C05456=1026.653,394.249,352.776,173.191,48.323,159.736
C05457=1026.645,394.003,352.820,173.181,48.321,159.734
C05458=1026.634,393.757,352.863,173.171,48.319,159.732
C05459=1026.625,393.511,352.907,173.161,48.317,159.730
C05460=1026.615,393.265,352.950,173.152,48.315,159.728
C05461=1026.606,393.019,352.994,173.141,48.312,159.726
C05462=1026.597,392.773,353.037,173.132,48.310,159.724
C05463=1026.586,392.527,353.080,173.121,48.309,159.722
C05464=1026.578,392.281,353.123,173.112,48.307,159.720
C05465=1026.568,392.035,353.167,173.102,48.304,159.718
C05466=1026.558,391.789,353.209,173.092,48.303,159.716
C05467=1026.549,391.543,353.253,173.082,48.301,159.714
C05468=1026.539,391.297,353.296,173.073,48.299,159.712
C05469=1026.530,391.051,353.338,173.063,48.297,159.711
C05470=1026.521,390.805,353.382,173.053,48.295,159.709
C05471=1026.511,390.559,353.425,173.044,48.293,159.707
C05472=1026.502,390.312,353.468,173.034,48.291,159.705
C05473=1026.493,390.067,353.511,173.024,48.289,159.703
C05474=1026.483,389.821,353.554,173.014,48.287,159.701
C05475=1026.474,389.575,353.597,173.005,48.285,159.699
C05476=1026.465,389.329,353.640,172.996,48.283,159.697
C05477=1026.455,389.083,353.683,172.987,48.282,159.696
C05478=1026.446,388.837,353.725,172.976,48.280,159.694
C05479=1026.437,388.590,353.768,172.967,48.278,159.692
C05480=1026.428,388.344,353.811,172.957,48.276,159.690
C05481=1026.418,388.097,353.853,172.948,48.275,159.688
C05482=1026.409,387.852,353.895,172.939,48.273,159.686
C05483=1026.400,387.606,353.938,172.930,48.271,159.685
C05484=1026.391,387.360,353.981,172.920,48.269,159.683
C05485=1026.381,387.113,354.024,172.910,48.268,159.681
C05486=1026.372,386.867,354.065,172.901,48.266,159.679
C05487=1026.363,386.621,354.108,172.892,48.264,159.677
C05488=1026.354,386.376,354.150,172.883,48.263,159.676
C05489=1026.344,386.128,354.192,172.873,48.261,159.674
C05490=1026.335,385.883,354.235,172.864,48.259,159.672
C05491=1026.326,385.636,354.276,172.855,48.258,159.671
C05492=1026.317,385.391,354.319,172.846,48.256,159.669
C05493=1026.307,385.144,354.361,172.837,48.255,159.667
C05494=1026.299,384.897,354.403,172.828,48.253,159.665
C05495=1026.289,384.651,354.445,172.818,48.252,159.664
C05496=1026.280,384.405,354.487,172.809,48.250,159.662
C05497=1026.271,384.159,354.528,172.800,48.248,159.660
C05498=1026.262,383.913,354.571,172.791,48.247,159.659
C05499=1026.253,383.667,354.613,172.782,48.245,159.657
C05500=1026.244,383.420,354.654,172.773,48.244,159.655
C05501=1026.235,383.174,354.696,172.764,48.242,159.654
C05502=1026.226,382.927,354.738,172.755,48.241,159.652
C05503=1026.218,382.681,354.779,172.746,48.240,159.650
C05504=1026.209,382.435,354.821,172.737,48.238,159.649
C05505=1026.199,382.189,354.862,172.728,48.237,159.647
C05506=1026.190,381.942,354.904,172.719,48.235,159.645
C05507=1026.181,381.696,354.946,172.710,48.234,159.644
C05508=1026.172,381.456,354.987,172.702,48.233,159.642
C05509=1026.163,381.216,355.028,172.693,48.231,159.641
C05510=1026.155,380.976,355.068,172.684,48.230,159.639
C05511=1026.146,380.736,355.109,172.676,48.229,159.638
C05512=1026.138,380.496,355.149,172.667,48.227,159.636
C05513=1026.129,380.257,355.189,172.659,48.226,159.634
C05514=1026.120,380.017,355.230,172.650,48.225,159.633
C05515=1026.112,379.776,355.270,172.641,48.223,159.631
C05516=1026.104,379.530,355.311,172.632,48.222,159.630
C05517=1026.095,379.284,355.353,172.624,48.220,159.628
C05518=1026.086,379.037,355.394,172.616,48.220,159.627
C05519=1026.077,378.790,355.435,172.607,48.218,159.625
C05520=1026.068,378.545,355.476,172.598,48.217,159.623
C05521=1026.059,378.298,355.517,172.590,48.216,159.622
C05522=1026.051,378.052,355.559,172.581,48.214,159.620
C05523=1026.042,377.805,355.600,172.572,48.213,159.619
C05524=1026.034,377.559,355.641,172.564,48.212,159.617
C05525=1026.025,377.312,355.682,172.555,48.211,159.616
C05526=1026.017,377.066,355.724,172.547,48.210,159.614
C05527=1026.008,376.819,355.765,172.539,48.208,159.613
C05528=1025.999,376.573,355.805,172.530,48.207,159.611
C05529=1025.990,376.327,355.846,172.521,48.206,159.610
C05530=1025.982,376.080,355.887,172.512,48.205,159.608
C05531=1025.972,375.833,355.928,172.505,48.204,159.607
C05532=1025.964,375.587,355.968,172.496,48.203,159.605
C05533=1025.955,375.340,356.009,172.488,48.201,159.604
C05534=1025.947,375.094,356.049,172.479,48.201,159.602
C05535=1025.937,374.847,356.090,172.470,48.200,159.601
C05536=1025.929,374.601,356.131,172.463,48.199,159.600
C05537=1025.921,374.354,356.172,172.454,48.198,159.598
C05538=1025.912,374.108,356.212,172.445,48.197,159.597
C05539=1025.903,373.861,356.253,172.438,48.196,159.595
C05540=1025.895,373.615,356.293,172.429,48.195,159.594
C05541=1025.886,373.368,356.334,172.421,48.193,159.592
C05542=1025.877,373.122,356.374,172.413,48.193,159.591
C05543=1025.869,372.875,356.415,172.405,48.191,159.589
C05544=1025.861,372.628,356.455,172.396,48.191,159.588
C05545=1025.852,372.382,356.495,172.388,48.190,159.587
C05546=1025.844,372.135,356.536,172.380,48.189,159.585
C05547=1025.835,371.889,356.576,172.371,48.188,159.584
C05548=1025.827,371.642,356.616,172.364,48.187,159.583
C05549=1025.818,371.396,356.656,172.355,48.187,159.581
C05550=1025.810,371.149,356.697,172.348,48.185,159.580
C05551=1025.802,370.903,356.737,172.340,48.184,159.578
C05552=1025.793,370.656,356.777,172.331,48.184,159.577
C05553=1025.785,370.409,356.817,172.324,48.183,159.576
C05554=1025.776,370.163,356.857,172.315,48.182,159.574
C05555=1025.768,369.916,356.897,172.308,48.181,159.573
C05556=1025.760,369.670,356.937,172.299,48.180,159.572
C05557=1025.751,369.423,356.977,172.292,48.180,159.571
C05558=1025.743,369.176,357.018,172.283,48.179,159.569
C05559=1025.735,368.930,357.057,172.276,48.178,159.568
C05560=1025.727,368.683,357.097,172.268,48.177,159.566
C05561=1025.718,368.437,357.137,172.259,48.177,159.565
C05562=1025.710,368.190,357.176,172.252,48.176,159.564
C05563=1025.701,367.943,357.216,172.243,48.175,159.563
C05564=1025.693,367.696,357.256,172.236,48.175,159.561
C05565=1025.685,367.449,357.295,172.228,48.173,159.560
C05566=1025.676,367.203,357.335,172.220,48.173,159.559
C05567=1025.668,366.956,357.374,172.213,48.173,159.558
C05568=1025.660,366.727,357.411,172.205,48.172,159.556
C05569=1025.652,366.498,357.448,172.198,48.171,159.555
C05570=1025.645,366.269,357.485,172.190,48.171,159.554
C05571=1025.637,366.039,357.521,172.183,48.170,159.553
C05572=1025.629,365.809,357.558,172.176,48.170,159.552
C05573=1025.622,365.580,357.595,172.169,48.170,159.551
C05574=1025.614,365.351,357.631,172.162,48.169,159.549
C05575=1025.607,365.122,357.668,172.155,48.168,159.548
C05576=1025.598,364.875,357.707,172.147,48.168,159.547
C05577=1025.590,364.629,357.747,172.139,48.167,159.546
C05578=1025.582,364.381,357.785,172.132,48.166,159.545
C05579=1025.573,364.135,357.825,172.124,48.166,159.543
C05580=1025.566,363.888,357.864,172.116,48.166,159.542
C05581=1025.557,363.641,357.904,172.109,48.165,159.541
C05582=1025.549,363.394,357.942,172.101,48.164,159.540
C05583=1025.540,363.147,357.982,172.094,48.164,159.539
C05584=1025.533,362.901,358.022,172.086,48.163,159.537
C05585=1025.525,362.654,358.060,172.079,48.163,159.536
C05586=1025.517,362.407,358.099,172.071,48.163,159.535
C05587=1025.509,362.160,358.138,172.064,48.162,159.534
C05588=1025.500,361.914,358.177,172.056,48.161,159.533
C05589=1025.493,361.666,358.216,172.048,48.161,159.531
C05590=1025.485,361.420,358.255,172.041,48.161,159.530
C05591=1025.477,361.173,358.294,172.034,48.160,159.529
C05592=1025.468,360.926,358.333,172.026,48.160,159.528
C05593=1025.460,360.679,358.372,172.019,48.159,159.527
C05594=1025.453,360.433,358.411,172.012,48.159,159.526
C05595=1025.445,360.186,358.450,172.004,48.159,159.525
C05596=1025.437,359.939,358.489,171.997,48.159,159.524
C05597=1025.428,359.691,358.527,171.989,48.158,159.522
C05598=1025.421,359.445,358.566,171.982,48.158,159.521
C05599=1025.412,359.198,358.605,171.975,48.158,159.520
C05600=1025.404,358.951,358.643,171.968,48.158,159.519
C05601=1025.397,358.705,358.682,171.959,48.157,159.518
C05602=1025.388,358.458,358.720,171.952,48.157,159.517
C05603=1025.380,358.210,358.758,171.945,48.157,159.516
C05604=1025.372,357.964,358.796,171.938,48.157,159.515
C05605=1025.364,357.717,358.835,171.931,48.157,159.514
C05606=1025.356,357.470,358.873,171.924,48.156,159.513
C05607=1025.348,357.223,358.912,171.916,48.156,159.512
C05608=1025.340,356.976,358.951,171.909,48.156,159.511
C05609=1025.333,356.729,358.989,171.902,48.155,159.509
C05610=1025.324,356.482,359.027,171.895,48.155,159.508
C05611=1025.317,356.235,359.066,171.888,48.155,159.507
C05612=1025.308,355.989,359.104,171.880,48.155,159.506
C05613=1025.301,355.741,359.141,171.873,48.155,159.505
C05614=1025.293,355.494,359.180,171.866,48.155,159.504
C05615=1025.285,355.248,359.218,171.859,48.155,159.503
C05616=1025.277,355.000,359.257,171.852,48.155,159.502
C05617=1025.270,354.753,359.294,171.844,48.155,159.501
C05618=1025.262,354.506,359.333,171.837,48.155,159.500
C05619=1025.253,354.260,359.370,171.830,48.155,159.499
C05620=1025.246,354.013,359.408,171.823,48.155,159.498
C05621=1025.238,353.766,359.447,171.816,48.155,159.497
C05622=1025.230,353.519,359.484,171.809,48.155,159.496
C05623=1025.222,353.272,359.522,171.802,48.155,159.495
C05624=1025.214,353.024,359.560,171.795,48.154,159.494
C05625=1025.206,352.778,359.597,171.788,48.154,159.493
C05626=1025.198,352.530,359.635,171.781,48.154,159.492
C05627=1025.191,352.284,359.673,171.774,48.154,159.491
C05628=1025.183,352.058,359.708,171.768,48.155,159.490
C05629=1025.176,351.832,359.742,171.761,48.155,159.489
C05630=1025.170,351.606,359.777,171.755,48.154,159.488
C05631=1025.162,351.380,359.811,171.749,48.155,159.488
C05632=1025.155,351.154,359.846,171.743,48.155,159.487
C05633=1025.147,350.928,359.880,171.737,48.155,159.486
C05634=1025.141,350.702,359.914,171.730,48.155,159.485
C05635=1025.134,350.476,359.949,171.724,48.155,159.484
C05636=1025.126,350.229,359.986,171.717,48.155,159.483
C05637=1025.119,349.982,360.024,171.710,48.155,159.482
C05638=1025.111,349.734,360.061,171.704,48.156,159.481
C05639=1025.103,349.488,360.099,171.696,48.156,159.480
C05640=1025.096,349.241,360.137,171.689,48.155,159.479
C05641=1025.088,348.993,360.174,171.683,48.156,159.479
C05642=1025.080,348.747,360.211,171.676,48.156,159.478
C05643=1025.073,348.499,360.249,171.670,48.156,159.477
C05644=1025.065,348.252,360.286,171.663,48.156,159.476
C05645=1025.057,348.005,360.323,171.656,48.156,159.475
C05646=1025.050,347.758,360.361,171.649,48.157,159.474
C05647=1025.042,347.511,360.398,171.642,48.157,159.473
C05648=1025.035,347.264,360.435,171.636,48.157,159.472
C05649=1025.027,347.017,360.472,171.629,48.158,159.471
C05650=1025.019,346.769,360.509,171.622,48.158,159.470
C05651=1025.012,346.522,360.546,171.616,48.158,159.470
C05652=1025.004,346.275,360.583,171.609,48.158,159.469
C05653=1024.997,346.028,360.621,171.602,48.159,159.468
C05654=1024.988,345.781,360.658,171.596,48.159,159.467
C05655=1024.981,345.533,360.695,171.589,48.159,159.466
C05656=1024.973,345.286,360.732,171.582,48.160,159.465
C05657=1024.965,345.039,360.768,171.576,48.160,159.465
C05658=1024.958,344.792,360.805,171.570,48.161,159.464
C05659=1024.950,344.545,360.842,171.562,48.161,159.463
C05660=1024.943,344.297,360.879,171.556,48.161,159.462
C05661=1024.936,344.051,360.916,171.549,48.162,159.461
C05662=1024.928,343.804,360.953,171.543,48.162,159.460
C05663=1024.921,343.556,360.989,171.537,48.163,159.460
C05664=1024.913,343.310,361.026,171.530,48.162,159.459
C05665=1024.905,343.062,361.063,171.523,48.163,159.458
C05666=1024.898,342.815,361.100,171.517,48.163,159.457
C05667=1024.890,342.567,361.136,171.511,48.164,159.456
C05668=1024.883,342.320,361.172,171.504,48.164,159.455
C05669=1024.876,342.073,361.210,171.497,48.165,159.455
C05670=1024.868,341.825,361.246,171.491,48.165,159.454
C05671=1024.860,341.579,361.283,171.485,48.166,159.453
C05672=1024.854,341.332,361.320,171.478,48.166,159.452
C05673=1024.846,341.084,361.356,171.471,48.167,159.451
C05674=1024.838,340.837,361.392,171.466,48.167,159.451
C05675=1024.831,340.590,361.430,171.459,48.168,159.450
C05676=1024.824,340.343,361.465,171.452,48.168,159.449
C05677=1024.816,340.095,361.502,171.446,48.169,159.448
C05678=1024.809,339.848,361.538,171.440,48.169,159.448
C05679=1024.802,339.600,361.575,171.433,48.170,159.447
C05680=1024.794,339.353,361.612,171.427,48.171,159.446
C05681=1024.787,339.107,361.647,171.421,48.171,159.445
C05682=1024.779,338.859,361.684,171.414,48.172,159.445
C05683=1024.771,338.612,361.720,171.408,48.172,159.444
C05684=1024.764,338.365,361.756,171.401,48.173,159.443
C05685=1024.756,338.118,361.792,171.396,48.174,159.442
C05686=1024.749,337.870,361.828,171.389,48.174,159.442
C05687=1024.741,337.622,361.864,171.383,48.176,159.441
C05688=1024.735,337.395,361.898,171.377,48.176,159.440
C05689=1024.728,337.168,361.930,171.372,48.177,159.440
C05690=1024.721,336.940,361.964,171.366,48.177,159.439
C05691=1024.714,336.713,361.997,171.359,48.178,159.438
C05692=1024.708,336.485,362.030,171.354,48.178,159.438
C05693=1024.700,336.257,362.063,171.348,48.179,159.437
C05694=1024.694,336.030,362.096,171.343,48.179,159.436
C05695=1024.687,335.803,362.129,171.337,48.180,159.436
C05696=1024.680,335.555,362.164,171.331,48.181,159.435
C05697=1024.673,335.307,362.201,171.324,48.182,159.434
C05698=1024.666,335.061,362.237,171.319,48.182,159.434
C05699=1024.658,334.813,362.273,171.312,48.184,159.433
C05700=1024.651,334.565,362.309,171.306,48.184,159.432
C05701=1024.644,334.318,362.344,171.300,48.185,159.432
C05702=1024.636,334.071,362.381,171.293,48.186,159.431
C05703=1024.629,333.824,362.416,171.288,48.186,159.430
C05704=1024.622,333.576,362.452,171.281,48.187,159.429
C05705=1024.615,333.329,362.487,171.275,48.188,159.429
C05706=1024.607,333.081,362.523,171.270,48.189,159.428
C05707=1024.600,332.834,362.558,171.263,48.190,159.427
C05708=1024.592,332.587,362.594,171.258,48.190,159.427
C05709=1024.585,332.340,362.629,171.251,48.192,159.426
C05710=1024.578,332.093,362.665,171.245,48.193,159.426
C05711=1024.571,331.845,362.701,171.239,48.193,159.425
C05712=1024.563,331.598,362.735,171.233,48.194,159.424
C05713=1024.556,331.350,362.771,171.227,48.195,159.424
C05714=1024.549,331.103,362.806,171.221,48.196,159.423
C05715=1024.542,330.855,362.842,171.215,48.198,159.423
C05716=1024.535,330.607,362.877,171.209,48.198,159.422
C05717=1024.527,330.361,362.912,171.203,48.199,159.421
C05718=1024.520,330.113,362.948,171.197,48.200,159.421
C05719=1024.513,329.866,362.983,171.191,48.201,159.420
C05720=1024.506,329.618,363.018,171.185,48.202,159.419
C05721=1024.498,329.371,363.054,171.179,48.203,159.419
C05722=1024.491,329.124,363.089,171.174,48.204,159.418
C05723=1024.484,328.876,363.124,171.167,48.205,159.418
C05724=1024.477,328.628,363.160,171.161,48.206,159.417
C05725=1024.470,328.381,363.195,171.156,48.207,159.416
C05726=1024.463,328.134,363.229,171.149,48.208,159.416
C05727=1024.456,327.886,363.264,171.144,48.209,159.415
C05728=1024.448,327.638,363.300,171.138,48.210,159.415
C05729=1024.441,327.392,363.336,171.132,48.211,159.414
C05730=1024.435,327.144,363.371,171.126,48.212,159.414
C05731=1024.427,326.897,363.405,171.120,48.213,159.413
C05732=1024.419,326.649,363.440,171.114,48.215,159.412
C05733=1024.412,326.401,363.475,171.109,48.215,159.412
C05734=1024.405,326.154,363.509,171.103,48.217,159.411
C05735=1024.397,325.907,363.544,171.097,48.218,159.411
C05736=1024.390,325.659,363.579,171.091,48.219,159.410
C05737=1024.383,325.412,363.613,171.085,48.220,159.410
C05738=1024.375,325.165,363.648,171.079,48.222,159.409
C05739=1024.369,324.917,363.682,171.073,48.223,159.409
C05740=1024.361,324.670,363.717,171.068,48.224,159.408
C05741=1024.353,324.422,363.752,171.062,48.226,159.408
C05742=1024.347,324.174,363.786,171.056,48.227,159.407
C05743=1024.339,323.927,363.820,171.050,48.228,159.406
C05744=1024.332,323.680,363.855,171.045,48.229,159.406
C05745=1024.325,323.432,363.889,171.039,48.231,159.405
C05746=1024.318,323.185,363.924,171.034,48.232,159.405
C05747=1024.311,322.937,363.958,171.027,48.233,159.404
C05748=1024.304,322.707,363.990,171.022,48.235,159.404
C05749=1024.297,322.477,364.023,171.017,48.236,159.404
C05750=1024.290,322.248,364.054,171.011,48.237,159.403
C05751=1024.284,322.018,364.086,171.006,48.238,159.403
C05752=1024.277,321.788,364.119,171.001,48.240,159.402
C05753=1024.270,321.558,364.150,170.996,48.240,159.402
C05754=1024.264,321.328,364.182,170.991,48.242,159.401
C05755=1024.258,321.099,364.214,170.986,48.243,159.401
C05756=1024.251,320.851,364.248,170.980,48.245,159.400
C05757=1024.243,320.604,364.282,170.974,48.245,159.400
C05758=1024.236,320.356,364.316,170.968,48.247,159.399
C05759=1024.230,320.108,364.351,170.963,48.248,159.399
C05760=1024.222,319.861,364.385,170.957,48.250,159.398
C05761=1024.215,319.614,364.419,170.952,48.251,159.398
C05762=1024.208,319.366,364.453,170.946,48.252,159.397
C05763=1024.201,319.118,364.488,170.940,48.254,159.397
C05764=1024.194,318.871,364.522,170.935,48.256,159.397
C05765=1024.187,318.623,364.556,170.929,48.257,159.396
C05766=1024.180,318.375,364.590,170.924,48.258,159.396
C05767=1024.173,318.129,364.624,170.918,48.260,159.395
C05768=1024.167,317.881,364.659,170.912,48.261,159.395
C05769=1024.160,317.633,364.693,170.907,48.263,159.394
C05770=1024.152,317.385,364.726,170.901,48.264,159.394
C05771=1024.146,317.137,364.761,170.896,48.265,159.393
C05772=1024.138,316.890,364.795,170.890,48.267,159.393
C05773=1024.132,316.643,364.829,170.885,48.269,159.393
C05774=1024.125,316.396,364.863,170.880,48.270,159.392
C05775=1024.118,316.148,364.897,170.874,48.271,159.392
C05776=1024.111,315.900,364.931,170.868,48.273,159.391
C05777=1024.104,315.652,364.965,170.863,48.274,159.391
C05778=1024.098,315.405,364.999,170.857,48.276,159.390
C05779=1024.091,315.157,365.033,170.852,48.278,159.390
C05780=1024.083,314.910,365.066,170.846,48.279,159.390
C05781=1024.077,314.662,365.101,170.841,48.281,159.389
C05782=1024.070,314.415,365.134,170.836,48.282,159.389
C05783=1024.063,314.167,365.168,170.830,48.284,159.388
C05784=1024.056,313.919,365.202,170.825,48.285,159.388
C05785=1024.050,313.672,365.236,170.820,48.287,159.387
C05786=1024.043,313.425,365.270,170.814,48.288,159.387
C05787=1024.036,313.177,365.304,170.809,48.290,159.387
C05788=1024.030,312.930,365.338,170.804,48.291,159.386
C05789=1024.023,312.681,365.371,170.798,48.293,159.386
C05790=1024.016,312.434,365.404,170.793,48.295,159.385
C05791=1024.009,312.187,365.438,170.788,48.296,159.385
C05792=1024.003,311.939,365.472,170.783,48.298,159.385
C05793=1023.996,311.692,365.506,170.777,48.299,159.384
C05794=1023.989,311.444,365.540,170.771,48.301,159.384
C05795=1023.983,311.196,365.572,170.766,48.302,159.384
C05796=1023.976,310.948,365.607,170.760,48.304,159.383
C05797=1023.970,310.701,365.640,170.755,48.306,159.383
C05798=1023.962,310.454,365.674,170.750,48.307,159.382
C05799=1023.955,310.205,365.707,170.744,48.309,159.382
C05800=1023.949,309.958,365.740,170.740,48.311,159.382
C05801=1023.941,309.711,365.773,170.735,48.313,159.381
C05802=1023.935,309.463,365.806,170.728,48.315,159.381
C05803=1023.928,309.215,365.840,170.724,48.317,159.381
C05804=1023.920,308.967,365.872,170.718,48.319,159.380
C05805=1023.914,308.720,365.905,170.713,48.321,159.380
C05806=1023.907,308.472,365.939,170.708,48.322,159.380
C05807=1023.900,308.225,365.971,170.702,48.324,159.379
C05808=1023.893,307.997,366.001,170.697,48.326,159.379
C05809=1023.886,307.770,366.032,170.693,48.327,159.379
C05810=1023.880,307.543,366.062,170.689,48.330,159.379
C05811=1023.874,307.316,366.092,170.684,48.331,159.378
C05812=1023.868,307.089,366.122,170.678,48.333,159.378
C05813=1023.861,306.861,366.152,170.674,48.335,159.378
C05814=1023.855,306.634,366.183,170.669,48.336,159.377
C05815=1023.849,306.407,366.213,170.664,48.338,159.377
C05816=1023.842,306.159,366.246,170.659,48.340,159.377
C05817=1023.835,305.911,366.278,170.654,48.342,159.377
C05818=1023.827,305.664,366.312,170.648,48.344,159.376
C05819=1023.821,305.416,366.345,170.644,48.346,159.376
C05820=1023.814,305.169,366.377,170.639,48.347,159.376
C05821=1023.807,304.921,366.410,170.633,48.350,159.375
C05822=1023.801,304.673,366.443,170.628,48.352,159.375
C05823=1023.793,304.425,366.475,170.623,48.354,159.375
C05824=1023.787,304.177,366.508,170.617,48.356,159.375
C05825=1023.781,303.930,366.541,170.612,48.357,159.374
C05826=1023.773,303.682,366.573,170.608,48.360,159.374
C05827=1023.767,303.434,366.606,170.602,48.362,159.374
C05828=1023.760,303.186,366.639,170.597,48.364,159.373
C05829=1023.753,302.939,366.671,170.592,48.366,159.373
C05830=1023.747,302.691,366.704,170.587,48.368,159.373
C05831=1023.740,302.444,366.736,170.581,48.370,159.373
C05832=1023.733,302.195,366.769,170.577,48.372,159.372
C05833=1023.726,301.948,366.802,170.572,48.374,159.372
C05834=1023.719,301.701,366.834,170.567,48.376,159.372
C05835=1023.712,301.452,366.867,170.561,48.378,159.372
C05836=1023.706,301.205,366.900,170.557,48.380,159.371
C05837=1023.699,300.957,366.932,170.552,48.382,159.371
C05838=1023.692,300.709,366.965,170.547,48.384,159.371
C05839=1023.685,300.461,366.997,170.541,48.386,159.371
C05840=1023.679,300.214,367.029,170.536,48.388,159.370
C05841=1023.673,299.966,367.062,170.532,48.391,159.370
C05842=1023.666,299.719,367.094,170.527,48.393,159.370
C05843=1023.659,299.470,367.127,170.521,48.394,159.370
C05844=1023.653,299.222,367.159,170.516,48.397,159.369
C05845=1023.646,298.975,367.191,170.512,48.399,159.369
C05846=1023.640,298.727,367.224,170.507,48.401,159.369
C05847=1023.633,298.480,367.256,170.501,48.403,159.369
C05848=1023.626,298.231,367.289,170.496,48.406,159.369
C05849=1023.620,297.984,367.321,170.492,48.408,159.368
C05850=1023.613,297.736,367.354,170.487,48.409,159.368
C05851=1023.607,297.488,367.386,170.482,48.411,159.368
C05852=1023.600,297.241,367.418,170.476,48.414,159.368
C05853=1023.593,296.993,367.451,170.472,48.416,159.367
C05854=1023.587,296.745,367.483,170.467,48.418,159.367
C05855=1023.580,296.498,367.515,170.462,48.420,159.367
C05856=1023.574,296.249,367.547,170.458,48.422,159.367
C05857=1023.567,296.001,367.580,170.452,48.425,159.367
C05858=1023.561,295.753,367.611,170.447,48.427,159.366
C05859=1023.554,295.506,367.644,170.442,48.429,159.366
C05860=1023.547,295.258,367.676,170.438,48.431,159.366
C05861=1023.541,295.010,367.708,170.433,48.433,159.366
C05862=1023.535,294.763,367.741,170.427,48.436,159.366
C05863=1023.528,294.515,367.772,170.423,48.438,159.365
C05864=1023.522,294.267,367.804,170.418,48.440,159.365
C05865=1023.515,294.019,367.837,170.413,48.442,159.365
C05866=1023.509,293.771,367.869,170.408,48.445,159.365
C05867=1023.502,293.524,367.901,170.404,48.447,159.365
C05868=1023.497,293.305,367.929,170.399,48.450,159.365
C05869=1023.491,293.086,367.957,170.395,48.452,159.365
C05870=1023.485,292.868,367.985,170.391,48.454,159.364
C05871=1023.480,292.650,368.013,170.386,48.456,159.364
C05872=1023.473,292.430,368.041,170.383,48.458,159.364
C05873=1023.467,292.212,368.069,170.378,48.460,159.364
C05874=1023.462,291.994,368.097,170.373,48.462,159.364
C05875=1023.456,291.775,368.124,170.370,48.464,159.364
C05876=1023.450,291.527,368.156,170.365,48.467,159.364
C05877=1023.443,291.280,368.188,170.359,48.469,159.363
C05878=1023.437,291.032,368.220,170.355,48.471,159.363
C05879=1023.430,290.784,368.251,170.350,48.474,159.363
C05880=1023.423,290.536,368.283,170.346,48.476,159.363
C05881=1023.416,290.288,368.314,170.341,48.478,159.363
C05882=1023.410,290.040,368.346,170.336,48.481,159.363
C05883=1023.403,289.792,368.377,170.331,48.483,159.363
C05884=1023.396,289.545,368.409,170.327,48.486,159.363
C05885=1023.390,289.297,368.440,170.322,48.488,159.362
C05886=1023.384,289.048,368.472,170.317,48.491,159.362
C05887=1023.377,288.801,368.503,170.312,48.494,159.362
C05888=1023.370,288.553,368.535,170.307,48.497,159.362
C05889=1023.363,288.305,368.566,170.303,48.499,159.362
C05890=1023.357,288.057,368.598,170.298,48.501,159.362
C05891=1023.351,287.810,368.629,170.294,48.504,159.362
C05892=1023.344,287.561,368.659,170.288,48.507,159.362
C05893=1023.337,287.313,368.691,170.284,48.509,159.361
C05894=1023.331,287.065,368.722,170.279,48.512,159.361
C05895=1023.324,286.817,368.754,170.275,48.514,159.361
C05896=1023.317,286.569,368.785,170.270,48.517,159.361
C05897=1023.311,286.321,368.816,170.265,48.519,159.361
C05898=1023.305,286.073,368.848,170.260,48.522,159.361
C05899=1023.299,285.826,368.879,170.256,48.525,159.361
C05900=1023.292,285.578,368.910,170.251,48.527,159.361
C05901=1023.285,285.330,368.942,170.247,48.530,159.361
C05902=1023.278,285.082,368.972,170.242,48.533,159.361
C05903=1023.271,284.834,369.003,170.237,48.535,159.361
C05904=1023.266,284.586,369.034,170.232,48.538,159.361
C05905=1023.259,284.338,369.065,170.228,48.541,159.361
C05906=1023.252,284.090,369.097,170.223,48.543,159.361
C05907=1023.246,283.841,369.127,170.219,48.546,159.360
C05908=1023.238,283.594,369.158,170.214,48.548,159.360
C05909=1023.232,283.346,369.189,170.209,48.552,159.360
C05910=1023.226,283.098,369.220,170.205,48.554,159.360
C05911=1023.219,282.850,369.251,170.200,48.557,159.360
C05912=1023.213,282.602,369.282,170.196,48.559,159.360
C05913=1023.207,282.354,369.312,170.191,48.562,159.360
C05914=1023.199,282.106,369.343,170.186,48.565,159.360
C05915=1023.193,281.858,369.374,170.182,48.568,159.360
C05916=1023.186,281.610,369.405,170.177,48.571,159.360
C05917=1023.180,281.362,369.436,170.173,48.574,159.360
C05918=1023.174,281.114,369.467,170.168,48.576,159.360
C05919=1023.166,280.866,369.497,170.164,48.579,159.360
C05920=1023.161,280.618,369.528,170.158,48.582,159.360
C05921=1023.154,280.370,369.559,170.154,48.585,159.360
C05922=1023.147,280.122,369.590,170.150,48.587,159.360
C05923=1023.142,279.874,369.620,170.145,48.590,159.360
C05924=1023.135,279.626,369.652,170.141,48.593,159.360
C05925=1023.128,279.378,369.682,170.137,48.596,159.360
C05926=1023.122,279.130,369.712,170.132,48.599,159.360
C05927=1023.115,278.882,369.744,170.127,48.602,159.360
C05928=1023.110,278.669,369.770,170.123,48.604,159.360
C05929=1023.104,278.457,369.796,170.120,48.606,159.360
C05930=1023.099,278.245,369.822,170.115,48.609,159.360
C05931=1023.093,278.032,369.848,170.112,48.611,159.360
C05932=1023.088,277.820,369.875,170.108,48.614,159.360
C05933=1023.083,277.608,369.901,170.104,48.616,159.359
C05934=1023.077,277.396,369.927,170.101,48.619,159.360
C05935=1023.071,277.182,369.953,170.096,48.621,159.360
C05936=1023.065,276.934,369.984,170.092,48.624,159.360
C05937=1023.058,276.686,370.014,170.088,48.627,159.360
C05938=1023.052,276.438,370.044,170.083,48.630,159.360
C05939=1023.045,276.190,370.074,170.079,48.633,159.360
C05940=1023.039,275.943,370.105,170.074,48.637,159.360
C05941=1023.032,275.695,370.135,170.069,48.639,159.360
C05942=1023.026,275.447,370.166,170.065,48.642,159.360
C05943=1023.020,275.198,370.197,170.061,48.645,159.360
C05944=1023.013,274.950,370.227,170.056,48.648,159.360
C05945=1023.007,274.702,370.257,170.052,48.651,159.360
C05946=1023.000,274.454,370.287,170.047,48.654,159.360
C05947=1022.994,274.206,370.317,170.043,48.657,159.360
C05948=1022.987,273.958,370.347,170.038,48.660,159.360
C05949=1022.981,273.710,370.377,170.034,48.664,159.360
C05950=1022.974,273.462,370.407,170.030,48.666,159.360
C05951=1022.968,273.214,370.438,170.026,48.669,159.360
C05952=1022.962,272.965,370.468,170.021,48.672,159.360
C05953=1022.955,272.718,370.498,170.016,48.676,159.360
C05954=1022.948,272.469,370.528,170.012,48.679,159.360
C05955=1022.942,272.222,370.559,170.007,48.681,159.360
C05956=1022.936,271.974,370.588,170.003,48.685,159.360
C05957=1022.930,271.725,370.618,169.999,48.688,159.360
C05958=1022.923,271.477,370.648,169.995,48.691,159.360
C05959=1022.917,271.229,370.679,169.991,48.694,159.360
C05960=1022.910,270.981,370.709,169.985,48.697,159.360
C05961=1022.904,270.732,370.739,169.981,48.701,159.360
C05962=1022.897,270.485,370.768,169.977,48.703,159.360
C05963=1022.892,270.237,370.799,169.973,48.707,159.361
C05964=1022.885,269.988,370.828,169.969,48.710,159.361
C05965=1022.878,269.741,370.858,169.965,48.713,159.361
C05966=1022.872,269.492,370.889,169.960,48.716,159.361
C05967=1022.866,269.244,370.918,169.955,48.720,159.361
C05968=1022.859,268.996,370.947,169.951,48.723,159.361
C05969=1022.853,268.748,370.978,169.947,48.726,159.361
C05970=1022.846,268.500,371.007,169.942,48.729,159.361
C05971=1022.839,268.252,371.037,169.938,48.732,159.361
C05972=1022.834,268.003,371.067,169.934,48.735,159.361
C05973=1022.827,267.756,371.097,169.930,48.739,159.361
C05974=1022.820,267.507,371.126,169.925,48.743,159.361
C05975=1022.814,267.259,371.156,169.921,48.745,159.361
C05976=1022.808,267.011,371.185,169.917,48.749,159.362
C05977=1022.801,266.763,371.216,169.912,48.752,159.362
C05978=1022.795,266.515,371.245,169.908,48.755,159.362
C05979=1022.789,266.267,371.275,169.904,48.759,159.362
C05980=1022.782,266.018,371.304,169.900,48.762,159.362
C05981=1022.776,265.770,371.334,169.895,48.765,159.362
C05982=1022.769,265.522,371.363,169.891,48.769,159.362
C05983=1022.763,265.274,371.392,169.887,48.772,159.362
C05984=1022.757,265.026,371.423,169.882,48.775,159.362
C05985=1022.750,264.777,371.452,169.878,48.779,159.362
C05986=1022.744,264.529,371.481,169.874,48.782,159.363
C05987=1022.737,264.281,371.511,169.869,48.786,159.363
C05988=1022.726,263.861,371.560,169.863,48.791,159.363
C05989=1022.721,263.651,371.585,169.859,48.794,159.363
C05990=1022.716,263.441,371.610,169.855,48.797,159.363
C05991=1022.710,263.231,371.635,169.852,48.800,159.363
C05992=1022.705,263.020,371.660,169.848,48.803,159.363
C05993=1022.699,262.810,371.685,169.845,48.806,159.363
C05994=1022.694,262.600,371.709,169.842,48.809,159.364
C05995=1022.687,262.352,371.739,169.836,48.812,159.364
C05996=1022.681,262.104,371.768,169.832,48.815,159.364
C05997=1022.676,261.856,371.798,169.828,48.819,159.364
C05998=1022.669,261.607,371.827,169.824,48.822,159.364
C05999=1022.663,261.359,371.856,169.820,48.826,159.364
C06000=1022.656,261.111,371.886,169.816,48.829,159.364
C06001=1022.650,260.863,371.915,169.812,48.833,159.365
C06002=1022.644,260.615,371.944,169.808,48.836,159.365
C06003=1022.637,260.366,371.973,169.803,48.840,159.365
C06004=1022.630,260.118,372.002,169.799,48.844,159.365
C06005=1022.624,259.870,372.032,169.795,48.847,159.365
C06006=1022.617,259.622,372.060,169.791,48.851,159.365
C06007=1022.611,259.374,372.089,169.787,48.854,159.366
C06008=1022.605,259.126,372.118,169.782,48.858,159.366
C06009=1022.597,258.877,372.146,169.778,48.861,159.366
C06010=1022.591,258.629,372.175,169.774,48.865,159.366
C06011=1022.585,258.380,372.204,169.770,48.869,159.366
C06012=1022.579,258.132,372.233,169.766,48.873,159.367
C06013=1022.572,257.884,372.262,169.761,48.876,159.367
C06014=1022.565,257.636,372.291,169.757,48.880,159.367
C06015=1022.559,257.387,372.319,169.753,48.883,159.367
C06016=1022.552,257.139,372.348,169.749,48.887,159.367
C06017=1022.546,256.891,372.377,169.746,48.891,159.368
C06018=1022.539,256.643,372.406,169.741,48.895,159.368
C06019=1022.533,256.395,372.435,169.737,48.898,159.368
C06020=1022.527,256.146,372.463,169.733,48.902,159.368
C06021=1022.520,255.898,372.492,169.729,48.906,159.368
C06022=1022.514,255.650,372.521,169.725,48.910,159.369
C06023=1022.507,255.402,372.549,169.720,48.913,159.369
C06024=1022.501,255.153,372.578,169.716,48.917,159.369
C06025=1022.494,254.905,372.607,169.712,48.921,159.369
C06026=1022.487,254.657,372.635,169.708,48.925,159.369
C06027=1022.481,254.408,372.664,169.704,48.928,159.370
C06028=1022.475,254.160,372.693,169.701,48.932,159.370
C06029=1022.469,253.912,372.722,169.696,48.936,159.370
C06030=1022.462,253.663,372.750,169.692,48.940,159.370
C06031=1022.456,253.415,372.779,169.688,48.943,159.370
C06032=1022.450,253.166,372.807,169.684,48.947,159.371
C06033=1022.443,252.919,372.835,169.680,48.951,159.371
C06034=1022.437,252.670,372.864,169.675,48.955,159.371
C06035=1022.431,252.422,372.893,169.671,48.959,159.371
C06036=1022.424,252.174,372.921,169.667,48.962,159.371
C06037=1022.418,251.925,372.950,169.664,48.966,159.372
C06038=1022.412,251.677,372.979,169.660,48.970,159.372
C06039=1022.405,251.429,373.006,169.656,48.973,159.372
C06040=1022.399,251.180,373.035,169.651,48.978,159.372
C06041=1022.393,250.932,373.064,169.647,48.981,159.373
C06042=1022.386,250.684,373.093,169.643,48.986,159.373
C06043=1022.380,250.435,373.120,169.639,48.989,159.373
C06044=1022.374,250.188,373.149,169.636,48.993,159.374
C06045=1022.368,249.939,373.177,169.632,48.997,159.374
C06046=1022.361,249.691,373.206,169.628,49.000,159.374
C06047=1022.356,249.480,373.230,169.624,49.004,159.374
C06048=1022.350,249.269,373.254,169.621,49.007,159.374
C06049=1022.345,249.058,373.279,169.617,49.011,159.374
C06050=1022.340,248.847,373.302,169.614,49.014,159.375
C06051=1022.334,248.637,373.327,169.611,49.017,159.375
C06052=1022.329,248.425,373.350,169.607,49.021,159.375
C06053=1022.324,248.215,373.375,169.604,49.024,159.375
C06054=1022.319,248.004,373.398,169.601,49.027,159.376
C06055=1022.313,247.756,373.427,169.596,49.031,159.376
C06056=1022.307,247.507,373.456,169.592,49.035,159.376
C06057=1022.301,247.258,373.484,169.588,49.039,159.376
C06058=1022.294,247.010,373.513,169.584,49.043,159.377
C06059=1022.288,246.761,373.541,169.581,49.047,159.377
C06060=1022.282,246.513,373.569,169.577,49.050,159.377
C06061=1022.275,246.266,373.597,169.573,49.055,159.377
C06062=1022.269,246.017,373.626,169.568,49.059,159.378
C06063=1022.264,245.768,373.654,169.564,49.063,159.378
C06064=1022.257,245.520,373.682,169.561,49.067,159.378
C06065=1022.251,245.272,373.711,169.557,49.070,159.378
C06066=1022.245,245.024,373.739,169.553,49.074,159.379
C06067=1022.239,244.775,373.766,169.549,49.079,159.379
C06068=1022.233,244.526,373.795,169.545,49.082,159.379
C06069=1022.226,244.278,373.824,169.541,49.087,159.380
C06070=1022.220,244.030,373.851,169.537,49.090,159.380
C06071=1022.214,243.782,373.879,169.533,49.094,159.380
C06072=1022.208,243.533,373.908,169.530,49.099,159.380
C06073=1022.202,243.284,373.936,169.526,49.103,159.381
C06074=1022.196,243.037,373.963,169.522,49.106,159.381
C06075=1022.190,242.788,373.991,169.518,49.110,159.381
C06076=1022.183,242.540,374.020,169.514,49.115,159.382
C06077=1022.176,242.292,374.047,169.510,49.119,159.382
C06078=1022.171,242.044,374.075,169.506,49.123,159.382
C06079=1022.164,241.795,374.103,169.502,49.127,159.382
C06080=1022.158,241.546,374.131,169.499,49.131,159.383
C06081=1022.151,241.298,374.159,169.494,49.136,159.383
C06082=1022.145,241.050,374.187,169.490,49.140,159.383
C06083=1022.140,240.801,374.214,169.487,49.144,159.384
C06084=1022.133,240.552,374.242,169.483,49.148,159.384
C06085=1022.128,240.304,374.270,169.479,49.152,159.385
C06086=1022.121,240.056,374.298,169.475,49.156,159.385
C06087=1022.114,239.808,374.325,169.471,49.160,159.385
C06088=1022.108,239.559,374.354,169.467,49.165,159.385
C06089=1022.102,239.311,374.381,169.463,49.169,159.386
C06090=1022.096,239.063,374.409,169.460,49.173,159.386
C06091=1022.089,238.814,374.436,169.456,49.177,159.386
C06092=1022.083,238.566,374.463,169.452,49.182,159.387
C06093=1022.076,238.317,374.491,169.448,49.186,159.387
C06094=1022.071,238.069,374.519,169.445,49.191,159.388
C06095=1022.064,237.821,374.546,169.441,49.195,159.388
C06096=1022.058,237.572,374.573,169.436,49.199,159.388
C06097=1022.051,237.323,374.601,169.433,49.204,159.389
C06098=1022.045,237.076,374.629,169.429,49.208,159.389
C06099=1022.039,236.827,374.656,169.425,49.212,159.389
C06100=1022.032,236.578,374.683,169.421,49.217,159.390
C06101=1022.026,236.330,374.711,169.417,49.221,159.390
C06102=1022.021,236.081,374.738,169.413,49.225,159.390
C06103=1022.014,235.833,374.766,169.410,49.230,159.391
C06104=1022.008,235.585,374.793,169.407,49.234,159.391
C06105=1022.001,235.336,374.820,169.402,49.239,159.391
C06106=1021.995,235.088,374.848,169.398,49.243,159.392
C06107=1021.989,234.874,374.871,169.396,49.247,159.392
C06108=1021.984,234.659,374.895,169.392,49.250,159.392
C06109=1021.978,234.446,374.918,169.389,49.254,159.393
C06110=1021.973,234.232,374.942,169.385,49.258,159.393
C06111=1021.968,234.017,374.966,169.381,49.262,159.393
C06112=1021.962,233.803,374.989,169.379,49.266,159.394
C06113=1021.957,233.589,375.012,169.375,49.269,159.394
C06114=1021.952,233.375,375.035,169.372,49.273,159.394
C06115=1021.945,233.127,375.063,169.369,49.277,159.395
C06116=1021.940,232.878,375.090,169.365,49.282,159.395
C06117=1021.933,232.630,375.118,169.361,49.287,159.396
C06118=1021.927,232.381,375.145,169.357,49.291,159.396
C06119=1021.921,232.133,375.172,169.353,49.295,159.396
C06120=1021.915,231.885,375.199,169.350,49.300,159.397
C06121=1021.908,231.636,375.227,169.345,49.305,159.397
C06122=1021.902,231.387,375.254,169.342,49.309,159.397
C06123=1021.896,231.139,375.281,169.339,49.314,159.398
C06124=1021.889,230.890,375.308,169.335,49.318,159.398
C06125=1021.884,230.642,375.335,169.330,49.323,159.399
C06126=1021.877,230.394,375.363,169.327,49.327,159.399
C06127=1021.871,230.145,375.389,169.323,49.332,159.399
C06128=1021.865,229.896,375.416,169.320,49.337,159.400
C06129=1021.859,229.648,375.444,169.315,49.341,159.400
C06130=1021.852,229.400,375.470,169.312,49.345,159.401
C06131=1021.846,229.151,375.497,169.309,49.350,159.401
C06132=1021.840,228.904,375.524,169.305,49.354,159.402
C06133=1021.833,228.655,375.551,169.301,49.360,159.402
C06134=1021.828,228.406,375.578,169.297,49.364,159.402
C06135=1021.821,228.158,375.605,169.294,49.369,159.403
C06136=1021.815,227.909,375.632,169.290,49.373,159.403
C06137=1021.809,227.660,375.659,169.286,49.378,159.404
C06138=1021.803,227.412,375.686,169.282,49.382,159.404
C06139=1021.796,227.164,375.713,169.279,49.387,159.405
C06140=1021.790,226.915,375.740,169.275,49.392,159.405
C06141=1021.784,226.667,375.766,169.271,49.397,159.405
C06142=1021.778,226.418,375.793,169.267,49.401,159.406
C06143=1021.771,226.170,375.819,169.264,49.406,159.406
C06144=1021.765,225.921,375.846,169.260,49.411,159.407
C06145=1021.759,225.673,375.873,169.256,49.415,159.407
C06146=1021.752,225.424,375.899,169.253,49.420,159.408
C06147=1021.746,225.175,375.926,169.249,49.425,159.408
C06148=1021.740,224.927,375.952,169.245,49.430,159.408
C06149=1021.733,224.678,375.979,169.242,49.435,159.409
C06150=1021.727,224.430,376.006,169.239,49.439,159.410
C06151=1021.720,224.181,376.032,169.234,49.445,159.410
C06152=1021.715,223.933,376.059,169.231,49.449,159.410
C06153=1021.709,223.684,376.085,169.227,49.454,159.411
C06154=1021.702,223.436,376.112,169.223,49.459,159.411
C06155=1021.696,223.187,376.139,169.219,49.463,159.412
C06156=1021.690,222.938,376.166,169.216,49.468,159.412
C06157=1021.683,222.690,376.192,169.212,49.473,159.413
C06158=1021.677,222.442,376.218,169.209,49.478,159.413
C06159=1021.670,222.193,376.245,169.205,49.483,159.414
C06160=1021.664,221.945,376.271,169.201,49.488,159.414
C06161=1021.659,221.696,376.298,169.198,49.493,159.415
C06162=1021.651,221.448,376.324,169.194,49.498,159.415
C06163=1021.646,221.199,376.351,169.191,49.503,159.416
C06164=1021.640,220.951,376.378,169.186,49.507,159.416
C06165=1021.633,220.702,376.404,169.183,49.512,159.416
C06166=1021.627,220.453,376.430,169.180,49.517,159.417
C06167=1021.621,220.236,376.453,169.176,49.521,159.417
C06168=1021.616,220.017,376.476,169.173,49.526,159.418
C06169=1021.611,219.799,376.500,169.170,49.530,159.418
C06170=1021.605,219.581,376.523,169.167,49.534,159.419
C06171=1021.600,219.363,376.547,169.163,49.538,159.419
C06172=1021.595,219.145,376.570,169.161,49.543,159.420
C06173=1021.589,218.927,376.592,169.157,49.547,159.420
C06174=1021.583,218.709,376.616,169.154,49.552,159.420
C06175=1021.578,218.460,376.642,169.150,49.556,159.421
C06176=1021.572,218.212,376.668,169.147,49.561,159.421
C06177=1021.565,217.964,376.694,169.143,49.567,159.422
C06178=1021.558,217.715,376.720,169.140,49.572,159.422
C06179=1021.552,217.466,376.746,169.136,49.576,159.423
C06180=1021.546,217.218,376.772,169.132,49.582,159.423
C06181=1021.540,216.969,376.798,169.129,49.587,159.424
C06182=1021.533,216.720,376.825,169.125,49.592,159.424
C06183=1021.527,216.472,376.851,169.122,49.597,159.425
C06184=1021.521,216.223,376.877,169.119,49.602,159.426
C06185=1021.515,215.975,376.903,169.114,49.608,159.426
C06186=1021.508,215.726,376.929,169.111,49.613,159.427
C06187=1021.502,215.477,376.955,169.108,49.617,159.427
C06188=1021.496,215.229,376.981,169.104,49.623,159.428
C06189=1021.490,214.981,377.007,169.100,49.628,159.428
C06190=1021.484,214.732,377.033,169.096,49.633,159.429
C06191=1021.477,214.483,377.059,169.093,49.638,159.429
C06192=1021.470,214.235,377.085,169.090,49.643,159.430
C06193=1021.465,213.986,377.111,169.086,49.649,159.430
C06194=1021.458,213.738,377.137,169.082,49.654,159.431
C06195=1021.452,213.489,377.162,169.079,49.659,159.431
C06196=1021.446,213.241,377.188,169.075,49.664,159.432
C06197=1021.440,212.992,377.215,169.072,49.669,159.432
C06198=1021.433,212.744,377.241,169.068,49.675,159.433
C06199=1021.427,212.495,377.266,169.065,49.680,159.434
C06200=1021.421,212.247,377.293,169.061,49.685,159.434
C06201=1021.415,211.998,377.318,169.057,49.690,159.435
C06202=1021.409,211.749,377.343,169.054,49.695,159.435
C06203=1021.403,211.501,377.370,169.050,49.701,159.436
C06204=1021.396,211.251,377.396,169.047,49.706,159.436
C06205=1021.390,211.003,377.422,169.044,49.711,159.437
C06206=1021.384,210.754,377.448,169.039,49.716,159.437
C06207=1021.378,210.506,377.474,169.036,49.721,159.438
C06208=1021.371,210.258,377.499,169.033,49.726,159.439
C06209=1021.366,210.009,377.525,169.029,49.732,159.439
C06210=1021.360,209.761,377.551,169.026,49.737,159.440
C06211=1021.353,209.512,377.576,169.022,49.742,159.440
C06212=1021.347,209.263,377.602,169.019,49.747,159.441
C06213=1021.341,209.015,377.627,169.015,49.753,159.441
C06214=1021.334,208.766,377.654,169.011,49.758,159.442
C06215=1021.328,208.517,377.679,169.009,49.764,159.443
C06216=1021.322,208.268,377.705,169.004,49.769,159.443
C06217=1021.316,208.020,377.730,169.001,49.774,159.444
C06218=1021.309,207.772,377.756,168.997,49.780,159.444
C06219=1021.303,207.523,377.782,168.994,49.785,159.445
C06220=1021.297,207.274,377.807,168.990,49.791,159.445
C06221=1021.291,207.026,377.832,168.987,49.796,159.446
C06222=1021.285,206.777,377.858,168.984,49.802,159.447
C06223=1021.278,206.529,377.884,168.980,49.807,159.447
C06224=1021.272,206.280,377.909,168.977,49.812,159.448
C06225=1021.266,206.031,377.934,168.973,49.818,159.448
C06226=1021.259,205.783,377.960,168.970,49.823,159.449
C06227=1021.254,205.567,377.982,168.967,49.828,159.450
C06228=1021.249,205.351,378.004,168.963,49.833,159.450
C06229=1021.243,205.135,378.026,168.961,49.837,159.451
C06230=1021.238,204.919,378.048,168.958,49.842,159.451
C06231=1021.232,204.704,378.070,168.954,49.847,159.452
C06232=1021.226,204.488,378.092,168.951,49.852,159.452
C06233=1021.221,204.272,378.114,168.948,49.857,159.453
C06234=1021.193,203.019,378.235,168.506,49.767,159.362
C06235=1021.188,202.770,378.258,168.502,49.773,159.363
C06236=1021.182,202.521,378.282,168.497,49.780,159.364
C06237=1021.177,202.272,378.306,168.492,49.786,159.364
C06238=1021.172,202.023,378.330,168.489,49.793,159.365
C06239=1021.166,201.774,378.353,168.484,49.799,159.365
C06240=1021.161,201.526,378.377,168.480,49.805,159.366
C06241=1021.156,201.277,378.401,168.475,49.812,159.367
C06242=1021.150,201.028,378.425,168.472,49.818,159.367
C06243=1021.145,200.779,378.448,168.467,49.825,159.368
C06244=1021.140,200.531,378.472,168.462,49.831,159.369
C06245=1021.135,200.281,378.496,168.458,49.838,159.369
C06246=1021.129,200.033,378.520,168.454,49.844,159.370
C06247=1021.124,199.784,378.543,168.450,49.851,159.371
C06248=1021.119,199.535,378.567,168.445,49.857,159.371
C06249=1021.113,199.286,378.590,168.442,49.864,159.372
C06250=1021.107,199.037,378.613,168.437,49.871,159.373
C06251=1021.102,198.788,378.637,168.432,49.877,159.373
C06252=1021.096,198.539,378.660,168.429,49.884,159.374
C06253=1021.091,198.291,378.684,168.424,49.890,159.374
C06254=1021.085,198.042,378.707,168.419,49.897,159.375
C06255=1021.080,197.793,378.730,168.416,49.904,159.376
C06256=1021.075,197.544,378.754,168.411,49.910,159.376
C06257=1021.069,197.295,378.776,168.407,49.917,159.377
C06258=1021.063,197.046,378.799,168.403,49.924,159.378
C06259=1021.058,196.797,378.824,168.399,49.930,159.379
C06260=1021.053,196.549,378.846,168.394,49.937,159.379
C06261=1021.047,196.300,378.869,168.390,49.944,159.380
C06262=1021.042,196.051,378.893,168.386,49.950,159.381
C06263=1021.036,195.802,378.916,168.381,49.957,159.381
C06264=1021.030,195.553,378.939,168.378,49.963,159.382
C06265=1021.025,195.304,378.962,168.373,49.970,159.383
C06266=1021.020,195.055,378.985,168.369,49.976,159.383
C06267=1021.015,194.806,379.009,168.365,49.983,159.384
C06268=1021.010,194.558,379.031,168.360,49.990,159.385
C06269=1021.004,194.309,379.054,168.356,49.996,159.385
C06270=1020.999,194.060,379.078,168.352,50.003,159.386
C06271=1020.993,193.811,379.101,168.348,50.010,159.387
C06272=1020.987,193.563,379.124,168.343,50.016,159.387
C06273=1020.982,193.313,379.148,168.340,50.023,159.388
C06274=1020.977,193.065,379.170,168.335,50.030,159.389
C06275=1020.972,192.816,379.193,168.331,50.036,159.389
C06276=1020.967,192.566,379.216,168.327,50.043,159.390
C06277=1020.961,192.318,379.239,168.323,50.050,159.391
C06278=1020.955,192.069,379.262,168.318,50.056,159.391
C06279=1020.951,191.820,379.285,168.315,50.063,159.392
C06280=1020.945,191.571,379.308,168.310,50.070,159.393
C06281=1020.939,191.322,379.331,168.307,50.076,159.394
C06282=1020.934,191.073,379.355,168.302,50.083,159.394
C06283=1020.929,190.825,379.377,168.298,50.090,159.395
C06284=1020.923,190.576,379.400,168.295,50.096,159.396
C06285=1020.918,190.327,379.424,168.290,50.103,159.396
C06286=1020.913,190.078,379.447,168.287,50.109,159.397
C06287=1020.908,189.829,379.469,168.282,50.116,159.398
C06288=1020.903,189.580,379.492,168.278,50.122,159.398
C06289=1020.897,189.331,379.515,168.274,50.129,159.399
C06290=1020.892,189.083,379.538,168.270,50.136,159.400
C06291=1020.887,188.834,379.561,168.267,50.143,159.401
C06292=1020.881,188.585,379.584,168.262,50.149,159.401
C06293=1020.876,188.336,379.606,168.258,50.156,159.402
C06294=1020.871,188.087,379.630,168.254,50.163,159.403
C06295=1020.864,187.805,379.655,168.249,50.170,159.403
C06296=1020.859,187.524,379.681,168.245,50.178,159.404
C06297=1020.853,187.242,379.707,168.241,50.185,159.405
C06298=1020.847,186.961,379.733,168.235,50.193,159.406
C06299=1020.842,186.713,379.756,168.232,50.199,159.406
C06300=1020.837,186.463,379.778,168.228,50.206,159.407
C06301=1020.832,186.214,379.801,168.224,50.212,159.408
C06302=1020.826,185.966,379.824,168.220,50.219,159.409
C06303=1020.821,185.716,379.847,168.217,50.226,159.409
C06304=1020.817,185.468,379.869,168.212,50.232,159.410
C06305=1020.811,185.219,379.892,168.208,50.239,159.411
C06306=1020.806,184.969,379.916,168.204,50.246,159.411
C06307=1020.801,184.721,379.938,168.200,50.253,159.412
C06308=1020.795,184.472,379.961,168.196,50.259,159.413
C06309=1020.791,184.223,379.984,168.192,50.266,159.413
C06310=1020.785,183.974,380.006,168.188,50.273,159.414
C06311=1020.780,183.726,380.029,168.184,50.279,159.415
C06312=1020.775,183.476,380.051,168.180,50.286,159.415
C06313=1020.771,183.228,380.074,168.177,50.292,159.416
C06314=1020.765,182.979,380.097,168.173,50.299,159.417
C06315=1020.759,182.729,380.119,168.169,50.305,159.418
C06316=1020.755,182.481,380.142,168.165,50.312,159.418
C06317=1020.750,182.231,380.165,168.161,50.319,159.419
C06318=1020.744,181.982,380.188,168.158,50.326,159.420
C06319=1020.739,181.733,380.209,168.153,50.333,159.421
C06320=1020.733,181.484,380.231,168.150,50.339,159.421
C06321=1020.728,181.235,380.253,168.145,50.347,159.422
C06322=1020.722,180.986,380.276,168.142,50.353,159.423
C06323=1020.717,180.738,380.297,168.137,50.360,159.424
C06324=1020.711,180.488,380.319,168.134,50.367,159.424
C06325=1020.706,180.239,380.342,168.129,50.374,159.425
C06326=1020.700,179.991,380.364,168.126,50.381,159.426
C06327=1020.695,179.741,380.386,168.122,50.388,159.427
C06328=1020.690,179.493,380.408,168.118,50.395,159.427
C06329=1020.684,179.243,380.429,168.115,50.401,159.428
C06330=1020.679,178.995,380.451,168.110,50.409,159.429
C06331=1020.673,178.745,380.473,168.107,50.415,159.430
C06332=1020.667,178.497,380.495,168.103,50.422,159.430
C06333=1020.662,178.248,380.518,168.099,50.429,159.431
C06334=1020.657,177.999,380.539,168.095,50.436,159.432
C06335=1020.652,177.749,380.562,168.091,50.444,159.433
C06336=1020.646,177.501,380.583,168.088,50.450,159.434
C06337=1020.641,177.251,380.605,168.084,50.457,159.434
C06338=1020.636,177.003,380.627,168.080,50.464,159.435
C06339=1020.630,176.754,380.649,168.076,50.471,159.436
C06340=1020.625,176.505,380.671,168.073,50.478,159.437
C06341=1020.619,176.256,380.693,168.068,50.485,159.437
C06342=1020.614,176.007,380.715,168.065,50.492,159.438
C06343=1020.608,175.758,380.737,168.060,50.499,159.439
C06344=1020.603,175.509,380.758,168.057,50.506,159.440
C06345=1020.598,175.260,380.780,168.054,50.512,159.440
C06346=1020.592,175.011,380.802,168.049,50.519,159.441
C06347=1020.587,174.762,380.824,168.046,50.526,159.442
C06348=1020.581,174.513,380.846,168.042,50.533,159.443
C06349=1020.577,174.264,380.868,168.038,50.540,159.443
C06350=1020.571,174.015,380.889,168.034,50.547,159.444
C06351=1020.566,173.766,380.911,168.031,50.554,159.445
C06352=1020.561,173.517,380.933,168.027,50.560,159.446
C06353=1020.555,173.268,380.955,168.023,50.567,159.446
C06354=1020.550,173.019,380.977,168.019,50.574,159.447
C06355=1020.545,172.770,380.998,168.016,50.581,159.448
C06356=1020.539,172.521,381.020,168.012,50.589,159.449
C06357=1020.534,172.272,381.042,168.009,50.596,159.450
C06358=1020.529,172.023,381.064,168.005,50.602,159.450
C06359=1020.523,171.741,381.088,168.001,50.610,159.451
C06360=1020.517,171.459,381.113,167.997,50.618,159.452
C06361=1020.511,171.177,381.137,167.992,50.626,159.453
C06362=1020.505,170.896,381.162,167.988,50.634,159.454
C06363=1020.499,170.646,381.184,167.984,50.641,159.455
C06364=1020.494,170.398,381.206,167.981,50.647,159.455
C06365=1020.490,170.149,381.228,167.978,50.654,159.456
C06366=1020.484,169.899,381.248,167.973,50.661,159.457
C06367=1020.479,169.650,381.270,167.970,50.668,159.458
C06368=1020.473,169.402,381.292,167.966,50.675,159.458
C06369=1020.468,169.152,381.314,167.963,50.682,159.459
C06370=1020.463,168.903,381.336,167.958,50.689,159.460
C06371=1020.458,168.655,381.357,167.955,50.696,159.461
C06372=1020.453,168.405,381.378,167.952,50.703,159.461
C06373=1020.448,168.156,381.400,167.948,50.709,159.462
C06374=1020.442,167.907,381.422,167.945,50.716,159.463
C06375=1020.437,167.659,381.443,167.940,50.723,159.464
C06376=1020.432,167.410,381.465,167.937,50.730,159.464
C06377=1020.427,167.160,381.486,167.933,50.737,159.465
C06378=1020.422,166.911,381.508,167.930,50.744,159.466
C06379=1020.416,166.663,381.529,167.927,50.750,159.467
C06380=1020.411,166.414,381.551,167.923,50.757,159.468
C06381=1020.406,166.164,381.573,167.919,50.764,159.468
C06382=1020.401,165.915,381.594,167.915,50.771,159.469
C06383=1020.396,165.666,381.616,167.912,50.778,159.470
C06384=1020.391,165.417,381.637,167.909,50.785,159.471
C06385=1020.386,165.168,381.658,167.905,50.792,159.471
C06386=1020.380,164.919,381.681,167.902,50.798,159.472
C06387=1020.375,164.670,381.702,167.897,50.806,159.473
C06388=1020.370,164.421,381.723,167.894,50.812,159.474
C06389=1020.365,164.172,381.745,167.891,50.819,159.474
C06390=1020.360,163.924,381.766,167.887,50.826,159.475
C06391=1020.355,163.674,381.787,167.884,50.833,159.476
C06392=1020.350,163.425,381.809,167.880,50.840,159.477
C06393=1020.345,163.176,381.830,167.877,50.847,159.478
C06394=1020.340,162.927,381.852,167.874,50.853,159.478
C06395=1020.334,162.678,381.873,167.869,50.861,159.479
C06396=1020.330,162.429,381.894,167.866,50.867,159.480
C06397=1020.325,162.180,381.916,167.862,50.874,159.481
C06398=1020.319,161.932,381.937,167.859,50.881,159.481
C06399=1020.314,161.681,381.959,167.856,50.888,159.482
C06400=1020.309,161.433,381.981,167.852,50.895,159.483
C06401=1020.304,161.183,382.001,167.849,50.902,159.484
C06402=1020.299,160.935,382.023,167.845,50.908,159.485
C06403=1020.294,160.685,382.044,167.842,50.915,159.485
C06404=1020.289,160.437,382.066,167.839,50.922,159.486
C06405=1020.285,160.188,382.088,167.835,50.929,159.487
C06406=1020.279,159.939,382.108,167.832,50.936,159.488
C06407=1020.274,159.690,382.130,167.828,50.943,159.488
C06408=1020.269,159.441,382.150,167.824,50.950,159.489
C06409=1020.264,159.192,382.172,167.821,50.957,159.490
C06410=1020.260,158.943,382.194,167.817,50.963,159.491
C06411=1020.254,158.693,382.214,167.814,50.970,159.492
C06412=1020.248,158.444,382.236,167.811,50.978,159.493
C06413=1020.243,158.195,382.256,167.808,50.985,159.493
C06414=1020.239,157.946,382.277,167.804,50.991,159.494
C06415=1020.233,157.697,382.299,167.801,50.998,159.495
C06416=1020.228,157.448,382.319,167.796,51.005,159.496
C06417=1020.223,157.199,382.340,167.793,51.013,159.497
C06418=1020.217,156.950,382.360,167.790,51.020,159.497
C06419=1020.212,156.701,382.382,167.787,51.027,159.498
C06420=1020.207,156.452,382.403,167.783,51.034,159.499
C06421=1020.202,156.203,382.423,167.780,51.041,159.500
C06422=1020.197,155.954,382.444,167.777,51.048,159.501
C06423=1020.191,155.672,382.468,167.773,51.056,159.502
C06424=1020.184,155.389,382.491,167.769,51.064,159.502
C06425=1020.178,155.107,382.515,167.765,51.072,159.503
C06426=1020.172,154.825,382.539,167.761,51.080,159.504
C06427=1020.167,154.575,382.559,167.758,51.087,159.505
C06428=1020.162,154.326,382.580,167.755,51.094,159.506
C06429=1020.157,154.077,382.601,167.751,51.101,159.507
C06430=1020.151,153.828,382.621,167.747,51.108,159.507
C06431=1020.147,153.579,382.642,167.744,51.115,159.508
C06432=1020.142,153.330,382.663,167.741,51.122,159.509
C06433=1020.136,153.080,382.683,167.737,51.129,159.510
C06434=1020.131,152.832,382.705,167.734,51.136,159.511
C06435=1020.126,152.583,382.725,167.731,51.143,159.512
C06436=1020.120,152.334,382.746,167.728,51.151,159.513
C06437=1020.115,152.085,382.766,167.724,51.157,159.513
C06438=1020.110,151.835,382.787,167.721,51.164,159.514
C06439=1020.104,151.586,382.807,167.718,51.171,159.515
C06440=1020.099,151.337,382.828,167.714,51.179,159.516
C06441=1020.094,151.088,382.848,167.710,51.186,159.517
C06442=1020.089,150.839,382.869,167.707,51.193,159.517
C06443=1020.084,150.590,382.889,167.704,51.200,159.518
C06444=1020.079,150.341,382.910,167.701,51.207,159.519
C06445=1020.074,150.092,382.930,167.697,51.214,159.520
C06446=1020.068,149.843,382.951,167.694,51.221,159.521
C06447=1020.063,149.593,382.971,167.691,51.228,159.521
C06448=1020.058,149.344,382.991,167.687,51.235,159.522
C06449=1020.053,149.095,383.012,167.684,51.242,159.523
C06450=1020.048,148.846,383.032,167.681,51.249,159.524
C06451=1020.042,148.597,383.053,167.678,51.256,159.525
C06452=1020.037,148.348,383.073,167.674,51.263,159.526
C06453=1020.032,148.099,383.094,167.671,51.271,159.527
C06454=1020.027,147.849,383.115,167.668,51.278,159.527
C06455=1020.021,147.601,383.135,167.665,51.285,159.528
C06456=1020.016,147.352,383.155,167.660,51.292,159.529
C06457=1020.011,147.103,383.175,167.657,51.299,159.530
C06458=1020.006,146.853,383.195,167.654,51.306,159.531
C06459=1020.000,146.604,383.216,167.651,51.313,159.531
C06460=1019.995,146.355,383.236,167.647,51.320,159.532
C06461=1019.990,146.106,383.257,167.645,51.328,159.533
C06462=1019.985,145.856,383.277,167.641,51.335,159.534
C06463=1019.980,145.607,383.297,167.638,51.341,159.535
C06464=1019.974,145.359,383.317,167.635,51.349,159.536
C06465=1019.969,145.110,383.337,167.632,51.356,159.536
C06466=1019.964,144.860,383.357,167.628,51.363,159.537
C06467=1019.959,144.611,383.378,167.625,51.370,159.538
C06468=1019.953,144.362,383.398,167.622,51.377,159.539
C06469=1019.948,144.112,383.418,167.619,51.384,159.540
C06470=1019.943,143.863,383.438,167.616,51.392,159.541
C06471=1019.937,143.615,383.458,167.613,51.399,159.542
C06472=1019.932,143.366,383.477,167.609,51.406,159.542
C06473=1019.927,143.116,383.498,167.606,51.413,159.543
C06474=1019.922,142.867,383.519,167.603,51.420,159.544
C06475=1019.916,142.618,383.538,167.599,51.427,159.545
C06476=1019.911,142.369,383.558,167.596,51.435,159.546
C06477=1019.907,142.120,383.578,167.592,51.442,159.547
C06478=1019.901,141.871,383.598,167.589,51.449,159.547
C06479=1019.895,141.622,383.618,167.586,51.456,159.548
C06480=1019.890,141.372,383.638,167.583,51.463,159.549
C06481=1019.884,141.123,383.658,167.580,51.470,159.550
C06482=1019.880,140.874,383.678,167.576,51.477,159.551
C06483=1019.875,140.625,383.698,167.573,51.485,159.552
C06484=1019.869,140.376,383.719,167.570,51.492,159.552
C06485=1019.864,140.126,383.738,167.567,51.499,159.553
C06486=1019.859,139.878,383.758,167.564,51.506,159.554
C06487=1019.853,139.596,383.781,167.561,51.514,159.555
C06488=1019.847,139.313,383.803,167.557,51.522,159.556
C06489=1019.841,139.030,383.826,167.553,51.530,159.557
C06490=1019.835,138.748,383.849,167.549,51.538,159.558
C06491=1019.831,138.499,383.868,167.546,51.546,159.559
C06492=1019.825,138.250,383.888,167.543,51.552,159.560
C06493=1019.820,138.000,383.908,167.540,51.559,159.560
C06494=1019.815,137.751,383.929,167.537,51.567,159.561
C06495=1019.810,137.502,383.947,167.534,51.574,159.562
C06496=1019.804,137.253,383.968,167.530,51.581,159.563
C06497=1019.799,137.004,383.987,167.528,51.589,159.564
C06498=1019.794,136.754,384.007,167.524,51.596,159.565
C06499=1019.788,136.506,384.027,167.521,51.602,159.565
C06500=1019.783,136.256,384.047,167.518,51.610,159.566
C06501=1019.778,136.007,384.066,167.515,51.617,159.567
C06502=1019.773,135.758,384.086,167.511,51.624,159.568
C06503=1019.767,135.509,384.105,167.509,51.632,159.569
C06504=1019.762,135.259,384.125,167.505,51.639,159.570
C06505=1019.756,135.010,384.145,167.502,51.646,159.571
C06506=1019.752,134.761,384.164,167.499,51.653,159.572
C06507=1019.746,134.512,384.184,167.496,51.660,159.572
C06508=1019.741,134.263,384.204,167.493,51.668,159.573
C06509=1019.736,134.014,384.223,167.490,51.675,159.574
C06510=1019.730,133.765,384.242,167.487,51.682,159.575
C06511=1019.725,133.515,384.262,167.485,51.689,159.576
C06512=1019.720,133.267,384.282,167.481,51.696,159.577
C06513=1019.715,133.017,384.302,167.478,51.703,159.578
C06514=1019.709,132.768,384.321,167.475,51.711,159.579
C06515=1019.705,132.519,384.340,167.472,51.718,159.579
C06516=1019.699,132.270,384.360,167.469,51.724,159.580
C06517=1019.693,132.020,384.380,167.466,51.732,159.581
C06518=1019.689,131.771,384.399,167.463,51.739,159.582
C06519=1019.683,131.522,384.418,167.459,51.746,159.583
C06520=1019.679,131.273,384.438,167.457,51.754,159.584
C06521=1019.673,131.024,384.458,167.453,51.761,159.584
C06522=1019.668,130.774,384.478,167.450,51.768,159.585
C06523=1019.663,130.525,384.496,167.447,51.775,159.586
C06524=1019.658,130.276,384.516,167.444,51.782,159.587
C06525=1019.652,130.026,384.536,167.441,51.789,159.588
C06526=1019.647,129.778,384.554,167.438,51.797,159.589
C06527=1019.641,129.528,384.574,167.435,51.804,159.590
C06528=1019.636,129.278,384.593,167.432,51.812,159.591
C06529=1019.631,129.030,384.612,167.428,51.819,159.591
C06530=1019.626,128.780,384.632,167.426,51.826,159.592
C06531=1019.620,128.531,384.651,167.422,51.833,159.593
C06532=1019.615,128.282,384.670,167.420,51.841,159.594
C06533=1019.609,128.033,384.689,167.416,51.848,159.595
C06534=1019.604,127.784,384.708,167.413,51.855,159.596
C06535=1019.598,127.534,384.727,167.410,51.863,159.597
C06536=1019.593,127.285,384.746,167.407,51.870,159.597
C06537=1019.588,127.036,384.765,167.404,51.877,159.598
C06538=1019.582,126.787,384.784,167.401,51.884,159.599
C06539=1019.578,126.538,384.804,167.398,51.892,159.600
C06540=1019.572,126.288,384.823,167.395,51.899,159.601
C06541=1019.567,126.040,384.842,167.392,51.907,159.602
C06542=1019.561,125.790,384.861,167.389,51.914,159.603
C06543=1019.556,125.540,384.880,167.386,51.921,159.604
C06544=1019.551,125.291,384.899,167.383,51.928,159.605
C06545=1019.545,125.042,384.918,167.380,51.936,159.606
C06546=1019.540,124.793,384.937,167.378,51.943,159.606
C06547=1019.534,124.544,384.956,167.375,51.950,159.607
C06548=1019.529,124.295,384.975,167.372,51.957,159.608
C06549=1019.523,124.046,384.994,167.368,51.964,159.609
C06550=1019.519,123.796,385.012,167.366,51.972,159.610
C06551=1019.513,123.513,385.034,167.362,51.980,159.611
C06552=1019.507,123.231,385.056,167.358,51.988,159.612
C06553=1019.501,122.949,385.077,167.356,51.996,159.613
C06554=1019.495,122.666,385.099,167.352,52.005,159.614
C06555=1019.490,122.417,385.118,167.349,52.012,159.615
C06556=1019.485,122.168,385.137,167.346,52.019,159.616
C06557=1019.479,121.919,385.156,167.343,52.026,159.616
C06558=1019.474,121.670,385.175,167.340,52.034,159.617
C06559=1019.468,121.420,385.194,167.337,52.041,159.618
C06560=1019.463,121.171,385.212,167.334,52.049,159.619
C06561=1019.458,120.922,385.232,167.331,52.056,159.620
C06562=1019.453,120.673,385.251,167.328,52.062,159.621
C06563=1019.447,120.423,385.269,167.326,52.070,159.622
C06564=1019.442,120.174,385.288,167.322,52.077,159.623
C06565=1019.436,119.925,385.307,167.320,52.085,159.624
C06566=1019.431,119.676,385.326,167.316,52.092,159.624
C06567=1019.427,119.426,385.345,167.313,52.099,159.625
C06568=1019.422,119.177,385.364,167.310,52.107,159.626
C06569=1019.416,118.928,385.383,167.307,52.114,159.627
C06570=1019.411,118.679,385.402,167.304,52.121,159.628
C06571=1019.406,118.429,385.420,167.302,52.128,159.629
C06572=1019.400,118.180,385.440,167.299,52.135,159.630
C06573=1019.395,117.931,385.459,167.296,52.142,159.630
C06574=1019.390,117.681,385.477,167.293,52.150,159.631
C06575=1019.385,117.433,385.496,167.290,52.157,159.632
C06576=1019.380,117.184,385.515,167.287,52.164,159.633
C06577=1019.374,116.934,385.533,167.284,52.171,159.634
C06578=1019.369,116.685,385.552,167.282,52.178,159.635
C06579=1019.364,116.436,385.571,167.278,52.185,159.636
C06580=1019.359,116.186,385.590,167.276,52.193,159.637
C06581=1019.354,115.938,385.608,167.273,52.200,159.637
C06582=1019.348,115.688,385.628,167.269,52.207,159.638
C06583=1019.343,115.439,385.646,167.266,52.214,159.639
C06584=1019.338,115.189,385.666,167.264,52.221,159.640
C06585=1019.333,114.940,385.685,167.261,52.228,159.641
C06586=1019.328,114.691,385.703,167.258,52.235,159.642
C06587=1019.323,114.441,385.722,167.255,52.243,159.643
C06588=1019.318,114.192,385.740,167.252,52.250,159.643
C06589=1019.313,113.943,385.759,167.250,52.257,159.644
C06590=1019.307,113.694,385.778,167.247,52.264,159.645
C06591=1019.302,113.445,385.796,167.244,52.272,159.646
C06592=1019.297,113.196,385.815,167.241,52.279,159.647
C06593=1019.292,112.946,385.834,167.238,52.286,159.648
C06594=1019.287,112.697,385.853,167.235,52.293,159.649
C06595=1019.282,112.448,385.871,167.233,52.300,159.650
C06596=1019.276,112.198,385.890,167.230,52.307,159.650
C06597=1019.272,111.949,385.908,167.226,52.314,159.651
C06598=1019.266,111.700,385.927,167.224,52.322,159.652
C06599=1019.260,111.450,385.945,167.220,52.329,159.653
C06600=1019.256,111.201,385.963,167.218,52.337,159.654
C06601=1019.250,110.952,385.982,167.216,52.344,159.655
C06602=1019.245,110.702,386.001,167.212,52.351,159.656
C06603=1019.239,110.454,386.019,167.210,52.358,159.657
C06604=1019.235,110.205,386.037,167.207,52.366,159.657
C06605=1019.229,109.955,386.056,167.204,52.373,159.658
C06606=1019.224,109.706,386.075,167.201,52.380,159.659
C06607=1019.219,109.457,386.092,167.197,52.387,159.660
C06608=1019.213,109.207,386.111,167.196,52.395,159.661
C06609=1019.208,108.958,386.130,167.193,52.402,159.662
C06610=1019.203,108.709,386.147,167.190,52.410,159.663
C06611=1019.197,108.459,386.166,167.187,52.417,159.664
C06612=1019.192,108.210,386.183,167.184,52.424,159.665
C06613=1019.187,107.961,386.202,167.181,52.432,159.665
C06614=1019.182,107.712,386.220,167.178,52.439,159.667
C06615=1019.175,107.428,386.241,167.175,52.447,159.668
C06616=1019.169,107.146,386.261,167.172,52.456,159.669
C06617=1019.163,106.864,386.282,167.168,52.464,159.669
C06618=1019.157,106.582,386.302,167.166,52.472,159.670
C06619=1019.152,106.332,386.320,167.163,52.480,159.671
C06620=1019.147,106.082,386.339,167.160,52.487,159.672
C06621=1019.141,105.834,386.357,167.157,52.494,159.673
C06622=1019.136,105.585,386.375,167.154,52.502,159.674
C06623=1019.130,105.335,386.393,167.151,52.509,159.675
C06624=1019.125,105.086,386.411,167.148,52.516,159.676
C06625=1019.120,104.837,386.429,167.145,52.523,159.677
C06626=1019.115,104.587,386.447,167.143,52.531,159.678
C06627=1019.109,104.338,386.466,167.140,52.538,159.679
C06628=1019.104,104.089,386.484,167.137,52.546,159.680
C06629=1019.099,103.839,386.502,167.134,52.553,159.680
C06630=1019.094,103.590,386.519,167.131,52.560,159.681
C06631=1019.089,103.341,386.537,167.128,52.568,159.682
C06632=1019.083,103.091,386.555,167.126,52.574,159.683
C06633=1019.078,102.842,386.574,167.124,52.582,159.684
C06634=1019.073,102.592,386.592,167.120,52.589,159.685
C06635=1019.068,102.343,386.609,167.117,52.596,159.686
C06636=1019.062,102.095,386.628,167.115,52.604,159.687
C06637=1019.056,101.845,386.646,167.112,52.611,159.687
C06638=1019.052,101.596,386.664,167.109,52.618,159.688
C06639=1019.046,101.347,386.682,167.107,52.626,159.689
C06640=1019.041,101.097,386.700,167.104,52.633,159.690
C06641=1019.036,100.848,386.718,167.100,52.640,159.691
C06642=1019.031,100.599,386.736,167.098,52.648,159.692
C06643=1019.026,100.349,386.754,167.096,52.655,159.693
C06644=1019.020,100.100,386.772,167.093,52.662,159.694
C06645=1019.015,99.850,386.790,167.090,52.669,159.695
C06646=1019.010,99.601,386.808,167.087,52.677,159.695
C06647=1019.005,99.352,386.826,167.085,52.683,159.696
C06648=1018.999,99.103,386.843,167.082,52.691,159.697
C06649=1018.994,98.853,386.862,167.079,52.698,159.698
C06650=1018.989,98.604,386.879,167.076,52.706,159.699
C06651=1018.983,98.355,386.897,167.073,52.713,159.700
C06652=1018.978,98.106,386.915,167.070,52.721,159.701
C06653=1018.973,97.856,386.932,167.067,52.728,159.702
C06654=1018.968,97.607,386.950,167.065,52.736,159.703
C06655=1018.962,97.358,386.967,167.063,52.743,159.704
C06656=1018.956,97.108,386.985,167.060,52.750,159.705
C06657=1018.951,96.859,387.003,167.057,52.758,159.705
C06658=1018.946,96.610,387.021,167.054,52.765,159.706
C06659=1018.940,96.360,387.038,167.051,52.773,159.707
C06660=1018.936,96.111,387.056,167.048,52.780,159.708
C06661=1018.930,95.862,387.073,167.045,52.787,159.709
C06662=1018.925,95.613,387.091,167.043,52.794,159.710
C06663=1018.919,95.364,387.108,167.041,52.802,159.711
C06664=1018.914,95.113,387.126,167.037,52.809,159.712
C06665=1018.908,94.864,387.144,167.034,52.816,159.712
C06666=1018.903,94.615,387.161,167.032,52.824,159.713
C06667=1018.897,94.366,387.179,167.029,52.831,159.714
C06668=1018.893,94.116,387.197,167.027,52.839,159.715
C06669=1018.887,93.867,387.214,167.024,52.846,159.716
C06670=1018.882,93.618,387.232,167.021,52.853,159.717
C06671=1018.876,93.369,387.249,167.018,52.861,159.718
C06672=1018.872,93.119,387.267,167.015,52.868,159.719
C06673=1018.866,92.870,387.284,167.012,52.876,159.720
C06674=1018.861,92.621,387.302,167.010,52.883,159.721
C06675=1018.855,92.372,387.319,167.007,52.890,159.721
C06676=1018.851,92.122,387.337,167.005,52.898,159.722
C06677=1018.845,91.873,387.354,167.002,52.905,159.723
C06678=1018.840,91.623,387.372,166.999,52.912,159.724
C06679=1018.835,91.376,387.390,166.997,52.919,159.725
C06680=1018.829,91.129,387.407,166.994,52.926,159.726
C06681=1018.824,90.882,387.424,166.991,52.934,159.727
C06682=1018.819,90.636,387.442,166.988,52.941,159.727
C06683=1018.814,90.389,387.459,166.986,52.948,159.729
C06684=1018.808,90.143,387.476,166.983,52.955,159.729
C06685=1018.804,89.896,387.493,166.980,52.962,159.730
C06686=1018.798,89.649,387.510,166.978,52.969,159.731
C06687=1018.793,89.400,387.528,166.975,52.977,159.732
C06688=1018.788,89.150,387.545,166.972,52.984,159.733
C06689=1018.783,88.901,387.563,166.970,52.992,159.734
C06690=1018.777,88.652,387.580,166.967,52.999,159.735
C06691=1018.772,88.402,387.597,166.963,53.006,159.735
C06692=1018.766,88.153,387.615,166.962,53.014,159.737
C06693=1018.761,87.904,387.632,166.959,53.021,159.737
C06694=1018.756,87.654,387.649,166.956,53.029,159.738
C06695=1018.750,87.405,387.666,166.953,53.036,159.739
C06696=1018.745,87.156,387.682,166.951,53.044,159.740
C06697=1018.739,86.907,387.700,166.947,53.051,159.741
C06698=1018.734,86.657,387.717,166.945,53.059,159.742
C06699=1018.728,86.408,387.734,166.943,53.066,159.743
C06700=1018.723,86.158,387.751,166.940,53.074,159.744
C06701=1018.718,85.909,387.769,166.937,53.081,159.745
C06702=1018.712,85.659,387.786,166.935,53.089,159.746
C06703=1018.707,85.410,387.803,166.931,53.096,159.746
C06704=1018.702,85.161,387.820,166.928,53.103,159.747
C06705=1018.696,84.911,387.837,166.926,53.111,159.748
C06706=1018.691,84.662,387.855,166.924,53.118,159.749
C06707=1018.686,84.412,387.871,166.921,53.126,159.750
C06708=1018.680,84.163,387.888,166.918,53.133,159.751
C06709=1018.675,83.914,387.906,166.916,53.141,159.752
C06710=1018.670,83.664,387.923,166.913,53.148,159.753
C06711=1018.663,83.415,387.940,166.909,53.155,159.754
C06712=1018.658,83.166,387.956,166.908,53.162,159.755
C06713=1018.654,82.917,387.973,166.905,53.170,159.755
C06714=1018.648,82.668,387.991,166.902,53.177,159.756
C06715=1018.643,82.418,388.007,166.899,53.185,159.757
C06716=1018.638,82.168,388.024,166.896,53.192,159.758
C06717=1018.632,81.919,388.042,166.895,53.199,159.759
C06718=1018.627,81.670,388.059,166.892,53.207,159.760
C06719=1018.622,81.420,388.075,166.889,53.214,159.761
C06720=1018.616,81.171,388.093,166.886,53.222,159.762
C06721=1018.611,80.921,388.110,166.883,53.229,159.763
C06722=1018.606,80.672,388.127,166.881,53.236,159.764
C06723=1018.601,80.423,388.144,166.878,53.244,159.765
C06724=1018.596,80.174,388.161,166.875,53.251,159.765
C06725=1018.590,79.924,388.178,166.872,53.258,159.766
C06726=1018.584,79.675,388.195,166.870,53.266,159.767
C06727=1018.579,79.426,388.211,166.868,53.273,159.768
C06728=1018.574,79.176,388.228,166.865,53.280,159.769
C06729=1018.569,78.926,388.245,166.862,53.288,159.770
C06730=1018.564,78.678,388.262,166.859,53.295,159.771
C06731=1018.557,78.390,388.282,166.857,53.303,159.772
C06732=1018.552,78.102,388.301,166.854,53.312,159.773
C06733=1018.545,77.815,388.321,166.850,53.320,159.774
C06734=1018.540,77.527,388.340,166.848,53.329,159.775
C06735=1018.534,77.277,388.357,166.845,53.336,159.776
C06736=1018.529,77.028,388.374,166.842,53.343,159.776
C06737=1018.523,76.779,388.391,166.839,53.351,159.777
C06738=1018.518,76.529,388.408,166.836,53.358,159.778
C06739=1018.513,76.280,388.425,166.834,53.365,159.779
C06740=1018.507,76.030,388.442,166.832,53.373,159.780
C06741=1018.502,75.781,388.457,166.829,53.380,159.781
C06742=1018.497,75.532,388.474,166.826,53.388,159.782
C06743=1018.491,75.249,388.493,166.824,53.396,159.783
C06744=1018.485,74.967,388.512,166.820,53.404,159.784
C06745=1018.478,74.685,388.531,166.817,53.413,159.785
C06746=1018.472,74.403,388.550,166.814,53.421,159.786
C06747=1018.467,74.153,388.566,166.812,53.429,159.787
C06748=1018.461,73.904,388.583,166.809,53.436,159.788
C06749=1018.456,73.655,388.599,166.806,53.443,159.789
C06750=1018.451,73.405,388.616,166.803,53.451,159.790
C06751=1018.445,73.156,388.632,166.801,53.458,159.791
C06752=1018.440,72.906,388.649,166.798,53.465,159.791
C06753=1018.435,72.656,388.666,166.796,53.473,159.792
C06754=1018.429,72.408,388.682,166.793,53.481,159.793
C06755=1018.424,72.158,388.699,166.790,53.489,159.794
C06756=1018.419,71.909,388.716,166.787,53.496,159.795
C06757=1018.413,71.659,388.732,166.785,53.503,159.796
C06758=1018.408,71.410,388.748,166.783,53.511,159.797
C06759=1018.402,71.161,388.765,166.780,53.518,159.798
C06760=1018.397,70.911,388.781,166.777,53.525,159.798
C06761=1018.392,70.662,388.798,166.774,53.533,159.799
C06762=1018.387,70.413,388.814,166.772,53.540,159.800
C06763=1018.381,70.163,388.831,166.769,53.547,159.801
C06764=1018.376,69.913,388.847,166.767,53.555,159.802
C06765=1018.371,69.664,388.863,166.764,53.562,159.803
C06766=1018.366,69.415,388.880,166.761,53.569,159.804
C06767=1018.360,69.165,388.896,166.759,53.577,159.805
C06768=1018.355,68.916,388.913,166.756,53.584,159.806
C06769=1018.349,68.667,388.929,166.754,53.591,159.807
C06770=1018.344,68.417,388.946,166.751,53.599,159.807
C06771=1018.339,68.168,388.963,166.748,53.607,159.808
C06772=1018.333,67.918,388.978,166.746,53.613,159.809
C06773=1018.328,67.669,388.994,166.744,53.621,159.810
C06774=1018.323,67.419,389.011,166.741,53.629,159.811
C06775=1018.317,67.170,389.027,166.738,53.636,159.812
C06776=1018.312,66.921,389.044,166.735,53.644,159.813
C06777=1018.307,66.671,389.059,166.732,53.651,159.814
C06778=1018.301,66.421,389.076,166.730,53.658,159.815
C06779=1018.296,66.173,389.092,166.728,53.666,159.816
C06780=1018.291,65.923,389.109,166.725,53.673,159.816
C06781=1018.285,65.673,389.124,166.722,53.680,159.817
C06782=1018.279,65.424,389.141,166.719,53.688,159.818
C06783=1018.275,65.175,389.157,166.716,53.696,159.819
C06784=1018.269,64.926,389.173,166.714,53.702,159.820
C06785=1018.264,64.675,389.189,166.712,53.710,159.821
C06786=1018.258,64.427,389.205,166.709,53.718,159.822
C06787=1018.253,64.177,389.222,166.707,53.726,159.823
C06788=1018.248,63.927,389.238,166.704,53.733,159.824
C06789=1018.242,63.678,389.254,166.701,53.740,159.824
C06790=1018.237,63.429,389.270,166.699,53.748,159.826
C06791=1018.231,63.179,389.286,166.696,53.755,159.826
C06792=1018.226,62.930,389.302,166.693,53.762,159.827
C06793=1018.221,62.680,389.318,166.691,53.770,159.828
C06794=1018.215,62.430,389.334,166.688,53.777,159.829
C06795=1018.210,62.181,389.349,166.685,53.785,159.830
C06796=1018.204,61.932,389.366,166.682,53.793,159.831
C06797=1018.199,61.682,389.381,166.680,53.801,159.832
C06798=1018.193,61.433,389.397,166.677,53.808,159.833
C06799=1018.188,61.183,389.413,166.675,53.816,159.834
C06800=1018.182,60.935,389.429,166.673,53.823,159.834
C06801=1018.177,60.685,389.444,166.670,53.831,159.836
C06802=1018.171,60.435,389.460,166.667,53.838,159.836
C06803=1018.166,60.186,389.475,166.664,53.845,159.837
C06804=1018.160,59.936,389.492,166.662,53.853,159.838
C06805=1018.155,59.687,389.508,166.659,53.861,159.839
C06806=1018.149,59.438,389.524,166.657,53.869,159.840
C06807=1018.143,59.155,389.541,166.653,53.877,159.841
C06808=1018.137,58.873,389.559,166.651,53.886,159.842
C06809=1018.130,58.590,389.577,166.648,53.894,159.843
C06810=1018.124,58.308,389.595,166.644,53.902,159.844
C06811=1018.119,58.059,389.610,166.642,53.910,159.845
C06812=1018.114,57.809,389.626,166.640,53.917,159.846
C06813=1018.108,57.560,389.642,166.637,53.925,159.847
C06814=1018.103,57.310,389.657,166.634,53.933,159.848
C06815=1018.097,57.061,389.674,166.632,53.941,159.849
C06816=1018.092,56.812,389.689,166.629,53.948,159.849
C06817=1018.086,56.562,389.704,166.626,53.955,159.850
C06818=1018.081,56.313,389.720,166.624,53.963,159.851
C06819=1018.075,56.063,389.736,166.621,53.970,159.852
C06820=1018.070,55.814,389.751,166.618,53.978,159.853
C06821=1018.064,55.564,389.767,166.616,53.985,159.854
C06822=1018.059,55.315,389.783,166.614,53.993,159.855
C06823=1018.054,55.065,389.798,166.611,54.000,159.856
C06824=1018.048,54.816,389.814,166.608,54.008,159.857
C06825=1018.043,54.567,389.829,166.605,54.015,159.857
C06826=1018.038,54.316,389.846,166.602,54.022,159.858
C06827=1018.032,54.068,389.862,166.600,54.030,159.859
C06828=1018.027,53.818,389.877,166.598,54.037,159.860
C06829=1018.022,53.568,389.892,166.595,54.045,159.861
C06830=1018.016,53.319,389.908,166.593,54.053,159.862
C06831=1018.011,53.070,389.924,166.590,54.060,159.863
C06832=1018.005,52.820,389.939,166.587,54.067,159.864
C06833=1018.000,52.571,389.955,166.585,54.075,159.865
C06834=1017.994,52.321,389.971,166.582,54.083,159.865
C06835=1017.989,52.072,389.986,166.580,54.090,159.866
C06836=1017.983,51.822,390.001,166.577,54.097,159.867
C06837=1017.978,51.573,390.017,166.575,54.105,159.868
C06838=1017.972,51.323,390.033,166.572,54.112,159.869
C06839=1017.967,51.074,390.048,166.569,54.119,159.870
C06840=1017.962,50.825,390.063,166.566,54.127,159.871
C06841=1017.956,50.576,390.079,166.564,54.134,159.872
C06842=1017.952,50.326,390.095,166.562,54.142,159.873
C06843=1017.946,50.076,390.111,166.559,54.149,159.873
C06844=1017.941,49.827,390.126,166.556,54.156,159.874
C06845=1017.935,49.577,390.142,166.553,54.164,159.875
C06846=1017.930,49.328,390.157,166.552,54.171,159.876
C06847=1017.925,49.078,390.173,166.549,54.179,159.877
C06848=1017.920,48.829,390.188,166.546,54.186,159.878
C06849=1017.915,48.580,390.203,166.543,54.194,159.879
C06850=1017.909,48.330,390.219,166.541,54.201,159.879
C06851=1017.904,48.081,390.235,166.539,54.208,159.880
C06852=1017.898,47.831,390.250,166.536,54.216,159.881
C06853=1017.893,47.582,390.265,166.533,54.223,159.882
C06854=1017.888,47.333,390.280,166.530,54.230,159.883
C06855=1017.882,47.083,390.296,166.528,54.238,159.884
C06856=1017.877,46.834,390.312,166.526,54.245,159.885
C06857=1017.871,46.584,390.327,166.523,54.252,159.886
C06858=1017.866,46.335,390.343,166.520,54.260,159.886
C06859=1017.861,46.085,390.358,166.517,54.267,159.887
C06860=1017.856,45.835,390.373,166.514,54.274,159.888
C06861=1017.851,45.586,390.389,166.513,54.281,159.889
C06862=1017.846,45.337,390.404,166.510,54.289,159.890
C06863=1017.841,45.087,390.420,166.507,54.297,159.891
C06864=1017.835,44.838,390.436,166.504,54.304,159.892
C06865=1017.830,44.588,390.451,166.503,54.311,159.892
C06866=1017.825,44.339,390.466,166.500,54.318,159.893
C06867=1017.820,44.089,390.482,166.497,54.326,159.894
C06868=1017.814,43.839,390.497,166.494,54.333,159.895
C06869=1017.809,43.590,390.512,166.492,54.340,159.896
C06870=1017.804,43.341,390.528,166.489,54.347,159.897
C06871=1017.798,43.059,390.545,166.486,54.356,159.897
C06872=1017.792,42.776,390.562,166.484,54.364,159.898
C06873=1017.786,42.494,390.579,166.480,54.372,159.899
C06874=1017.780,42.211,390.597,166.478,54.380,159.900
C06875=1017.775,41.962,390.612,166.475,54.388,159.901
C06876=1017.769,41.712,390.627,166.473,54.396,159.902
C06877=1017.764,41.463,390.643,166.470,54.403,159.903
C06878=1017.758,41.214,390.657,166.467,54.410,159.904
C06879=1017.752,40.964,390.673,166.464,54.418,159.905
C06880=1017.748,40.714,390.687,166.463,54.425,159.906
C06881=1017.743,40.465,390.702,166.460,54.433,159.907
C06882=1017.736,40.215,390.717,166.457,54.440,159.907
C06883=1017.731,39.966,390.732,166.454,54.447,159.908
C06884=1017.726,39.716,390.748,166.452,54.455,159.909
C06885=1017.721,39.466,390.763,166.449,54.463,159.910
C06886=1017.715,39.217,390.778,166.446,54.470,159.911
C06887=1017.710,38.968,390.792,166.445,54.477,159.912
C06888=1017.705,38.718,390.807,166.442,54.485,159.913
C06889=1017.699,38.468,390.823,166.439,54.492,159.913
C06890=1017.694,38.219,390.838,166.436,54.499,159.914
C06891=1017.688,37.970,390.853,166.434,54.507,159.915
C06892=1017.683,37.721,390.868,166.431,54.515,159.916
C06893=1017.678,37.470,390.883,166.429,54.522,159.917
C06894=1017.672,37.221,390.897,166.426,54.529,159.918
C06895=1017.667,36.972,390.912,166.423,54.536,159.919
C06896=1017.662,36.722,390.928,166.421,54.544,159.919
C06897=1017.657,36.472,390.942,166.418,54.551,159.920
C06898=1017.651,36.223,390.957,166.416,54.559,159.921
C06899=1017.646,35.974,390.972,166.414,54.566,159.922
C06900=1017.640,35.724,390.986,166.411,54.574,159.923
C06901=1017.635,35.474,391.002,166.408,54.581,159.924
C06902=1017.629,35.225,391.016,166.406,54.589,159.925
C06903=1017.624,34.976,391.031,166.403,54.596,159.926
C06904=1017.618,34.726,391.046,166.400,54.604,159.926
C06905=1017.613,34.476,391.060,166.397,54.611,159.927
C06906=1017.608,34.227,391.075,166.395,54.619,159.928
C06907=1017.602,33.978,391.090,166.392,54.627,159.929
C06908=1017.597,33.728,391.104,166.389,54.634,159.930
C06909=1017.591,33.478,391.119,166.388,54.641,159.931
C06910=1017.586,33.229,391.133,166.385,54.648,159.932
C06911=1017.581,32.979,391.148,166.383,54.656,159.933
C06912=1017.575,32.730,391.163,166.380,54.664,159.933
C06913=1017.570,32.481,391.177,166.377,54.671,159.934
C06914=1017.564,32.231,391.192,166.374,54.679,159.935
C06915=1017.559,31.981,391.207,166.371,54.686,159.936
C06916=1017.553,31.732,391.221,166.369,54.693,159.937
C06917=1017.549,31.482,391.236,166.366,54.701,159.938
C06918=1017.543,31.233,391.250,166.364,54.708,159.939
C06919=1017.538,30.983,391.265,166.362,54.716,159.939
C06920=1017.532,30.734,391.280,166.359,54.723,159.940
C06921=1017.527,30.484,391.294,166.356,54.731,159.941
C06922=1017.521,30.235,391.309,166.353,54.738,159.942
C06923=1017.517,29.985,391.323,166.351,54.745,159.943
C06924=1017.511,29.736,391.338,166.348,54.753,159.943
C06925=1017.506,29.486,391.352,166.347,54.761,159.945
C06926=1017.500,29.237,391.367,166.344,54.768,159.945
C06927=1017.495,28.987,391.382,166.341,54.775,159.946
C06928=1017.489,28.738,391.396,166.338,54.783,159.947
C06929=1017.484,28.488,391.411,166.335,54.790,159.948
C06930=1017.479,28.239,391.425,166.333,54.798,159.949
C06931=1017.474,27.989,391.440,166.330,54.805,159.949
C06932=1017.468,27.740,391.454,166.328,54.812,159.950
C06933=1017.463,27.490,391.469,166.325,54.819,159.951
C06934=1017.458,27.240,391.483,166.323,54.827,159.952
C06935=1017.451,26.958,391.499,166.319,54.835,159.953
C06936=1017.445,26.675,391.516,166.316,54.844,159.954
C06937=1017.439,26.393,391.532,166.314,54.853,159.955
C06938=1017.433,26.111,391.548,166.311,54.861,159.956
C06939=1017.427,25.862,391.562,166.308,54.869,159.957
C06940=1017.422,25.612,391.577,166.305,54.876,159.957
C06941=1017.417,25.363,391.591,166.303,54.883,159.958
C06942=1017.411,25.113,391.605,166.300,54.891,159.959
C06943=1017.406,24.864,391.619,166.299,54.898,159.960
C06944=1017.401,24.614,391.633,166.296,54.906,159.961
C06945=1017.395,24.365,391.648,166.293,54.913,159.962
C06946=1017.390,24.115,391.662,166.290,54.921,159.963
C06947=1017.384,23.865,391.676,166.287,54.928,159.963
C06948=1017.379,23.615,391.690,166.285,54.936,159.964
C06949=1017.373,23.366,391.705,166.282,54.943,159.965
C06950=1017.368,23.116,391.719,166.279,54.950,159.966
C06951=1017.362,22.867,391.733,166.277,54.959,159.967
C06952=1017.357,22.617,391.747,166.274,54.966,159.968
C06953=1017.352,22.368,391.762,166.271,54.973,159.968
C06954=1017.346,22.118,391.776,166.269,54.981,159.969
C06955=1017.341,21.869,391.790,166.267,54.988,159.970
C06956=1017.336,21.619,391.804,166.264,54.995,159.971
C06957=1017.330,21.369,391.818,166.262,55.003,159.972
C06958=1017.325,21.120,391.832,166.259,55.010,159.973
C06959=1017.319,20.871,391.846,166.256,55.018,159.973
C06960=1017.314,20.621,391.860,166.253,55.025,159.974
C06961=1017.309,20.371,391.875,166.251,55.032,159.975
C06962=1017.304,20.122,391.888,166.248,55.040,159.976
C06963=1017.298,19.872,391.902,166.246,55.047,159.977
C06964=1017.293,19.623,391.916,166.243,55.054,159.978
C06965=1017.288,19.373,391.931,166.241,55.062,159.978
C06966=1017.282,19.124,391.945,166.238,55.069,159.979
C06967=1017.277,18.874,391.959,166.235,55.077,159.980
C06968=1017.271,18.625,391.973,166.233,55.085,159.981
C06969=1017.266,18.375,391.987,166.230,55.092,159.982
C06970=1017.260,18.126,392.001,166.227,55.100,159.983
C06971=1017.255,17.876,392.015,166.225,55.107,159.983
C06972=1017.249,17.626,392.028,166.222,55.114,159.984
C06973=1017.244,17.376,392.043,166.219,55.122,159.985
C06974=1017.239,17.127,392.057,166.217,55.129,159.986
C06975=1017.234,16.878,392.070,166.215,55.136,159.987
C06976=1017.229,16.628,392.084,166.212,55.144,159.988
C06977=1017.223,16.379,392.098,166.209,55.151,159.988
C06978=1017.218,16.129,392.112,166.207,55.159,159.989
C06979=1017.212,15.880,392.126,166.204,55.166,159.990
C06980=1017.207,15.630,392.140,166.201,55.174,159.991
C06981=1017.201,15.381,392.153,166.199,55.181,159.992
C06982=1017.196,15.131,392.167,166.196,55.189,159.992
C06983=1017.190,14.881,392.181,166.193,55.196,159.993
C06984=1017.185,14.632,392.195,166.190,55.203,159.994
C06985=1017.179,14.382,392.209,166.189,55.211,159.995
C06986=1017.175,14.132,392.223,166.186,55.218,159.996
C06987=1017.169,13.883,392.237,166.183,55.225,159.997
C06988=1017.164,13.634,392.251,166.181,55.233,159.997
C06989=1017.159,13.384,392.264,166.178,55.240,159.998
C06990=1017.154,13.134,392.278,166.175,55.248,159.999
C06991=1017.148,12.885,392.292,166.172,55.255,160.000
C06992=1017.142,12.635,392.305,166.170,55.263,160.001
C06993=1017.136,12.386,392.319,166.168,55.271,160.002
C06994=1017.131,12.136,392.332,166.165,55.278,160.002
C06995=1017.126,11.886,392.346,166.162,55.286,160.003
C06996=1017.120,11.636,392.360,166.159,55.293,160.004
C06997=1017.115,11.388,392.373,166.157,55.301,160.005
C06998=1017.110,11.138,392.386,166.154,55.308,160.006
C06999=1017.103,10.857,392.401,166.151,55.317,160.007
C07000=1017.097,10.575,392.417,166.148,55.325,160.007
C07001=1017.091,10.295,392.432,166.145,55.334,160.009
C07002=1017.085,10.014,392.447,166.142,55.342,160.009
C07003=1017.080,9.764,392.461,166.140,55.350,160.010
C07004=1017.073,9.515,392.474,166.137,55.357,160.011
C07005=1017.068,9.265,392.487,166.134,55.365,160.012
C07006=1017.063,9.016,392.500,166.132,55.373,160.013
C07007=1017.058,8.766,392.514,166.129,55.380,160.014
C07008=1017.053,8.516,392.527,166.127,55.388,160.015
C07009=1017.046,8.267,392.541,166.124,55.395,160.015
C07010=1017.041,8.017,392.555,166.121,55.403,160.016
C07011=1017.036,7.768,392.567,166.119,55.410,160.017
C07012=1017.031,7.518,392.581,166.116,55.418,160.018
C07013=1017.025,7.269,392.595,166.113,55.425,160.019
C07014=1017.020,7.019,392.608,166.111,55.433,160.019
C07015=1017.014,6.769,392.622,166.108,55.440,160.020
C07016=1017.009,6.520,392.634,166.105,55.448,160.021
C07017=1017.004,6.270,392.648,166.102,55.455,160.022
C07018=1016.998,6.021,392.661,166.101,55.462,160.023
C07019=1016.993,5.771,392.675,166.098,55.470,160.024
C07020=1016.988,5.522,392.688,166.096,55.477,160.024
C07021=1016.983,5.272,392.701,166.093,55.485,160.025
C07022=1016.976,5.022,392.715,166.090,55.491,160.026
C07023=1016.971,4.773,392.728,166.087,55.499,160.026
C07024=1016.966,4.523,392.741,166.084,55.506,160.027
C07025=1016.961,4.274,392.755,166.082,55.514,160.028
C07026=1016.956,4.023,392.768,166.079,55.521,160.029
C07027=1016.949,3.774,392.781,166.076,55.529,160.030
C07028=1016.945,3.525,392.794,166.074,55.536,160.031
C07029=1016.939,3.275,392.808,166.071,55.544,160.031
C07030=1016.934,3.025,392.821,166.068,55.551,160.032
C07031=1016.929,2.776,392.834,166.066,55.559,160.033
C07032=1016.923,2.526,392.847,166.063,55.566,160.033
C07033=1016.918,2.277,392.861,166.061,55.573,160.034
C07034=1016.913,2.026,392.874,166.058,55.580,160.035
C07035=1016.907,1.778,392.887,166.056,55.588,160.036
C07036=1016.902,1.528,392.900,166.053,55.595,160.037
C07037=1016.897,1.278,392.914,166.050,55.603,160.038
C07038=1016.892,1.029,392.927,166.048,55.610,160.038
C07039=1016.886,0.779,392.940,166.044,55.617,160.039
C07040=1016.881,0.529,392.953,166.042,55.625,160.040
C07041=1016.876,0.280,392.967,166.039,55.632,160.041
C07042=1016.871,0.030,392.980,166.037,55.640,160.041
C07043=1016.865,-0.220,392.994,166.035,55.647,160.042
C07044=1016.860,-0.469,393.006,166.032,55.653,160.043
C07045=1016.854,-0.718,393.020,166.029,55.661,160.044
C07046=1016.850,-0.968,393.033,166.027,55.668,160.045
C07047=1016.845,-1.218,393.046,166.024,55.676,160.045
C07048=1016.838,-1.467,393.059,166.021,55.683,160.046
C07049=1016.834,-1.717,393.072,166.018,55.690,160.047
C07050=1016.828,-1.966,393.086,166.015,55.698,160.048
C07051=1016.823,-2.216,393.099,166.014,55.705,160.049
C07052=1016.818,-2.466,393.111,166.011,55.712,160.049
C07053=1016.812,-2.715,393.125,166.008,55.719,160.050
C07054=1016.808,-2.965,393.138,166.005,55.727,160.051
C07055=1016.802,-3.214,393.152,166.002,55.734,160.051
C07056=1016.796,-3.464,393.164,166.000,55.741,160.052
C07057=1016.792,-3.714,393.177,165.997,55.749,160.053
C07058=1016.786,-3.963,393.191,165.995,55.756,160.054
C07059=1016.782,-4.213,393.204,165.992,55.762,160.054
C07060=1016.776,-4.463,393.216,165.990,55.770,160.055
C07061=1016.771,-4.713,393.229,165.987,55.778,160.056
C07062=1016.765,-4.961,393.242,165.984,55.785,160.057
C07063=1016.759,-5.241,393.257,165.981,55.794,160.058
C07064=1016.753,-5.519,393.271,165.978,55.802,160.058
C07065=1016.747,-5.798,393.285,165.976,55.810,160.059
C07066=1016.740,-6.077,393.299,165.972,55.819,160.060
C07067=1016.736,-6.327,393.312,165.970,55.826,160.061
C07068=1016.730,-6.577,393.325,165.967,55.833,160.062
C07069=1016.725,-6.826,393.337,165.964,55.840,160.062
C07070=1016.719,-7.076,393.350,165.961,55.848,160.063
C07071=1016.714,-7.326,393.362,165.959,55.856,160.064
C07072=1016.709,-7.576,393.375,165.956,55.863,160.065
C07073=1016.703,-7.825,393.388,165.954,55.871,160.066
C07074=1016.698,-8.075,393.400,165.951,55.878,160.066
C07075=1016.693,-8.325,393.413,165.948,55.885,160.067
C07076=1016.687,-8.574,393.425,165.945,55.893,160.068
C07077=1016.682,-8.824,393.439,165.943,55.900,160.069
C07078=1016.676,-9.073,393.451,165.940,55.908,160.069
C07079=1016.671,-9.323,393.464,165.937,55.915,160.070
C07080=1016.666,-9.572,393.477,165.934,55.922,160.071
C07081=1016.660,-9.822,393.489,165.932,55.930,160.072
C07082=1016.655,-10.071,393.501,165.929,55.937,160.072
C07083=1016.650,-10.321,393.515,165.927,55.945,160.073
C07084=1016.644,-10.571,393.527,165.924,55.952,160.074
C07085=1016.639,-10.821,393.540,165.921,55.959,160.075
C07086=1016.634,-11.070,393.552,165.918,55.967,160.075
C07087=1016.629,-11.319,393.564,165.916,55.974,160.076
C07088=1016.623,-11.569,393.577,165.913,55.982,160.077
C07089=1016.618,-11.819,393.590,165.911,55.988,160.078
C07090=1016.612,-12.068,393.602,165.908,55.996,160.079
C07091=1016.608,-12.318,393.615,165.906,56.003,160.079
C07092=1016.602,-12.568,393.627,165.903,56.010,160.080
C07093=1016.597,-12.817,393.640,165.900,56.018,160.081
C07094=1016.591,-13.067,393.653,165.898,56.025,160.082
C07095=1016.586,-13.317,393.664,165.894,56.032,160.082
C07096=1016.582,-13.566,393.677,165.892,56.040,160.083
C07097=1016.576,-13.816,393.690,165.889,56.047,160.084
C07098=1016.570,-14.066,393.702,165.886,56.054,160.084
C07099=1016.565,-14.316,393.715,165.884,56.061,160.085
C07100=1016.560,-14.565,393.727,165.881,56.069,160.086
C07101=1016.555,-14.814,393.739,165.878,56.076,160.086
C07102=1016.549,-15.064,393.752,165.876,56.083,160.087
C07103=1016.544,-15.313,393.765,165.874,56.091,160.088
C07104=1016.539,-15.564,393.778,165.871,56.097,160.089
C07105=1016.534,-15.813,393.789,165.868,56.105,160.090
C07106=1016.529,-16.063,393.801,165.865,56.112,160.090
C07107=1016.523,-16.313,393.814,165.862,56.119,160.091
C07108=1016.517,-16.562,393.826,165.860,56.127,160.092
C07109=1016.512,-16.812,393.839,165.857,56.135,160.093
C07110=1016.507,-17.062,393.851,165.855,56.142,160.093
C07111=1016.502,-17.311,393.863,165.852,56.149,160.094
C07112=1016.496,-17.561,393.876,165.849,56.157,160.095
C07113=1016.491,-17.811,393.887,165.847,56.164,160.095
C07114=1016.486,-18.060,393.899,165.844,56.172,160.096
C07115=1016.480,-18.310,393.912,165.841,56.179,160.097
C07116=1016.475,-18.559,393.923,165.838,56.186,160.098
C07117=1016.470,-18.809,393.935,165.836,56.194,160.098
C07118=1016.464,-19.058,393.948,165.833,56.201,160.099
C07119=1016.459,-19.308,393.959,165.830,56.208,160.100
C07120=1016.454,-19.558,393.972,165.828,56.216,160.101
C07121=1016.448,-19.808,393.985,165.825,56.223,160.101
C07122=1016.443,-20.057,393.996,165.822,56.230,160.102
C07123=1016.438,-20.307,394.008,165.819,56.238,160.103
C07124=1016.433,-20.556,394.020,165.817,56.245,160.104
C07125=1016.427,-20.806,394.033,165.814,56.252,160.104
C07126=1016.422,-21.055,394.045,165.811,56.260,160.105
C07127=1016.416,-21.333,394.058,165.808,56.268,160.106
C07128=1016.410,-21.609,394.071,165.806,56.276,160.107
C07129=1016.404,-21.887,394.084,165.802,56.284,160.107
C07130=1016.398,-22.164,394.098,165.798,56.292,160.108
C07131=1016.393,-22.414,394.110,165.796,56.300,160.109
C07132=1016.388,-22.663,394.122,165.794,56.307,160.110
C07133=1016.383,-22.913,394.134,165.791,56.314,160.110
C07134=1016.377,-23.163,394.146,165.789,56.321,160.111
C07135=1016.372,-23.413,394.158,165.786,56.328,160.112
C07136=1016.367,-23.662,394.170,165.783,56.336,160.112
C07137=1016.361,-23.911,394.182,165.780,56.343,160.113
C07138=1016.356,-24.162,394.194,165.778,56.350,160.114
C07139=1016.351,-24.411,394.206,165.775,56.358,160.115
C07140=1016.346,-24.661,394.218,165.772,56.365,160.115
C07141=1016.340,-24.910,394.230,165.769,56.372,160.116
C07142=1016.335,-25.160,394.241,165.766,56.379,160.117
C07143=1016.329,-25.410,394.254,165.764,56.387,160.117
C07144=1016.324,-25.659,394.265,165.761,56.394,160.118
C07145=1016.320,-25.909,394.278,165.758,56.401,160.119
C07146=1016.315,-26.159,394.290,165.755,56.408,160.119
C07147=1016.309,-26.408,394.302,165.754,56.415,160.120
C07148=1016.304,-26.658,394.314,165.751,56.422,160.121
C07149=1016.299,-26.908,394.325,165.748,56.430,160.122
C07150=1016.294,-27.157,394.337,165.745,56.437,160.122
C07151=1016.289,-27.407,394.349,165.742,56.444,160.123
C07152=1016.283,-27.656,394.361,165.739,56.451,160.123
C07153=1016.278,-27.907,394.373,165.736,56.458,160.124
C07154=1016.273,-28.157,394.384,165.734,56.466,160.125
C07155=1016.267,-28.406,394.396,165.731,56.473,160.126
C07156=1016.262,-28.655,394.407,165.728,56.480,160.126
C07157=1016.257,-28.905,394.419,165.726,56.488,160.127
C07158=1016.252,-29.155,394.430,165.723,56.496,160.128
C07159=1016.246,-29.404,394.443,165.720,56.502,160.128
C07160=1016.240,-29.654,394.454,165.718,56.510,160.129
C07161=1016.235,-29.904,394.465,165.715,56.517,160.130
C07162=1016.230,-30.154,394.477,165.712,56.525,160.131
C07163=1016.225,-30.404,394.488,165.710,56.532,160.131
C07164=1016.220,-30.653,394.500,165.707,56.539,160.132
C07165=1016.214,-30.902,394.511,165.704,56.547,160.133
C07166=1016.209,-31.152,394.523,165.701,56.554,160.133
C07167=1016.204,-31.402,394.534,165.699,56.561,160.134
C07168=1016.199,-31.652,394.546,165.696,56.568,160.135
C07169=1016.194,-31.901,394.558,165.693,56.576,160.135
C07170=1016.187,-32.151,394.569,165.690,56.583,160.136
C07171=1016.182,-32.401,394.581,165.688,56.590,160.137
C07172=1016.177,-32.651,394.592,165.684,56.597,160.137
C07173=1016.172,-32.901,394.603,165.682,56.605,160.138
C07174=1016.167,-33.150,394.614,165.679,56.612,160.139
C07175=1016.161,-33.399,394.627,165.676,56.619,160.139
C07176=1016.156,-33.649,394.638,165.673,56.626,160.140
C07177=1016.151,-33.899,394.649,165.671,56.634,160.141
C07178=1016.146,-34.149,394.661,165.668,56.641,160.141
C07179=1016.140,-34.398,394.672,165.665,56.648,160.142
C07180=1016.135,-34.648,394.683,165.662,56.655,160.143
C07181=1016.130,-34.898,394.695,165.660,56.662,160.143
C07182=1016.125,-35.147,394.706,165.658,56.670,160.144
C07183=1016.120,-35.397,394.717,165.655,56.676,160.145
C07184=1016.114,-35.646,394.729,165.652,56.684,160.146
C07185=1016.109,-35.896,394.741,165.649,56.691,160.146
C07186=1016.104,-36.146,394.752,165.646,56.698,160.147
C07187=1016.099,-36.395,394.763,165.644,56.706,160.147
C07188=1016.094,-36.645,394.775,165.641,56.712,160.148
C07189=1016.089,-36.895,394.786,165.638,56.720,160.149
C07190=1016.084,-37.145,394.798,165.635,56.727,160.149
C07191=1016.078,-37.421,394.810,165.633,56.735,160.150
C07192=1016.072,-37.697,394.823,165.629,56.743,160.151
C07193=1016.066,-37.973,394.835,165.627,56.750,160.152
C07194=1016.060,-38.249,394.847,165.623,56.758,160.152
C07195=1016.055,-38.498,394.859,165.620,56.765,160.153
C07196=1016.050,-38.748,394.870,165.617,56.772,160.153
C07197=1016.045,-38.998,394.882,165.615,56.780,160.154
C07198=1016.040,-39.248,394.893,165.613,56.786,160.155
C07199=1016.035,-39.497,394.904,165.610,56.793,160.155
C07200=1016.030,-39.747,394.916,165.607,56.801,160.156
C07201=1016.024,-39.997,394.926,165.604,56.808,160.157
C07202=1016.019,-40.247,394.937,165.602,56.816,160.158
C07203=1016.014,-40.497,394.948,165.599,56.823,160.158
C07204=1016.009,-40.746,394.959,165.596,56.830,160.159
C07205=1016.003,-40.995,394.970,165.593,56.837,160.159
C07206=1015.999,-41.246,394.981,165.590,56.844,160.160
C07207=1015.993,-41.495,394.992,165.588,56.852,160.161
C07208=1015.988,-41.745,395.003,165.585,56.859,160.161
C07209=1015.982,-41.994,395.014,165.583,56.866,160.162
C07210=1015.977,-42.244,395.026,165.580,56.873,160.163
C07211=1015.972,-42.494,395.036,165.577,56.880,160.163
C07212=1015.967,-42.744,395.047,165.574,56.888,160.164
C07213=1015.962,-42.993,395.058,165.571,56.895,160.165
C07214=1015.957,-43.243,395.069,165.569,56.903,160.165
C07215=1015.951,-43.493,395.079,165.566,56.909,160.166
C07216=1015.946,-43.743,395.091,165.563,56.916,160.167
C07217=1015.940,-43.992,395.102,165.560,56.924,160.167
C07218=1015.935,-44.242,395.112,165.557,56.931,160.168
C07219=1015.930,-44.492,395.123,165.554,56.938,160.168
C07220=1015.925,-44.741,395.134,165.552,56.946,160.169
C07221=1015.920,-44.991,395.145,165.549,56.953,160.170
C07222=1015.914,-45.241,395.155,165.546,56.960,160.170
C07223=1015.909,-45.490,395.167,165.543,56.966,160.171
C07224=1015.904,-45.740,395.178,165.540,56.974,160.172
C07225=1015.900,-45.990,395.188,165.538,56.981,160.172
C07226=1015.894,-46.239,395.199,165.535,56.988,160.173
C07227=1015.889,-46.489,395.211,165.532,56.995,160.173
C07228=1015.883,-46.739,395.221,165.530,57.002,160.174
C07229=1015.878,-46.989,395.232,165.527,57.009,160.175
C07230=1015.874,-47.238,395.242,165.524,57.016,160.175
C07231=1015.869,-47.488,395.253,165.521,57.023,160.176
C07232=1015.863,-47.738,395.264,165.519,57.031,160.177
C07233=1015.858,-47.988,395.275,165.516,57.038,160.177
C07234=1015.853,-48.237,395.286,165.513,57.045,160.178
C07235=1015.848,-48.487,395.297,165.511,57.051,160.179
C07236=1015.843,-48.737,395.307,165.508,57.058,160.179
C07237=1015.838,-48.987,395.319,165.505,57.065,160.180
C07238=1015.833,-49.236,395.328,165.502,57.073,160.180
C07239=1015.827,-49.485,395.339,165.499,57.080,160.181
C07240=1015.822,-49.736,395.350,165.496,57.087,160.181
C07241=1015.817,-49.985,395.361,165.493,57.094,160.182
C07242=1015.812,-50.234,395.372,165.490,57.101,160.183
C07243=1015.807,-50.485,395.382,165.488,57.107,160.183
C07244=1015.802,-50.735,395.393,165.486,57.114,160.184
C07245=1015.796,-50.984,395.404,165.483,57.121,160.184
C07246=1015.792,-51.234,395.414,165.480,57.129,160.185
C07247=1015.786,-51.484,395.425,165.477,57.136,160.186
C07248=1015.781,-51.734,395.435,165.474,57.143,160.186
C07249=1015.776,-51.984,395.445,165.472,57.150,160.187
C07250=1015.771,-52.233,395.455,165.469,57.157,160.188
C07251=1015.765,-52.483,395.466,165.466,57.165,160.188
C07252=1015.760,-52.733,395.476,165.463,57.172,160.189
C07253=1015.755,-52.982,395.486,165.460,57.179,160.189
C07254=1015.749,-53.232,395.497,165.458,57.187,160.190
C07255=1015.744,-53.505,395.508,165.454,57.194,160.191
C07256=1015.738,-53.779,395.519,165.452,57.202,160.191
C07257=1015.732,-54.052,395.530,165.448,57.210,160.192
C07258=1015.726,-54.325,395.542,165.445,57.218,160.193
C07259=1015.721,-54.575,395.552,165.442,57.225,160.193
C07260=1015.716,-54.824,395.562,165.439,57.233,160.194
C07261=1015.711,-55.075,395.572,165.436,57.240,160.195
C07262=1015.705,-55.324,395.583,165.433,57.247,160.195
C07263=1015.700,-55.573,395.592,165.432,57.254,160.196
C07264=1015.695,-55.824,395.603,165.429,57.261,160.197
C07265=1015.690,-56.074,395.613,165.426,57.268,160.197
C07266=1015.685,-56.323,395.623,165.423,57.275,160.198
C07267=1015.679,-56.573,395.634,165.421,57.283,160.199
C07268=1015.675,-56.822,395.644,165.418,57.290,160.199
C07269=1015.669,-57.072,395.654,165.415,57.297,160.200
C07270=1015.664,-57.322,395.664,165.412,57.304,160.200
C07271=1015.659,-57.572,395.674,165.409,57.311,160.201
C07272=1015.653,-57.822,395.684,165.406,57.318,160.201
C07273=1015.649,-58.071,395.694,165.404,57.325,160.202
C07274=1015.643,-58.322,395.704,165.401,57.332,160.203
C07275=1015.638,-58.570,395.715,165.398,57.339,160.203
C07276=1015.633,-58.820,395.725,165.395,57.346,160.204
C07277=1015.628,-59.070,395.735,165.392,57.353,160.204
C07278=1015.622,-59.320,395.745,165.389,57.360,160.205
C07279=1015.618,-59.569,395.755,165.386,57.367,160.205
C07280=1015.612,-59.819,395.765,165.384,57.375,160.206
C07281=1015.607,-60.069,395.774,165.382,57.382,160.207
